   // COMANDO DELLE USCITE SUL SOLLEVAMENTO RIBALTATORE
   // 
   REGION COMANDO DELLE USCITE SOLLEVATORE RIBALTA P3
       // Sollevatore Ribalta Semi guscio prodotto Stazione P3 - RIPOSO
       "A0301_CinghiaTrasporto_1.1_V_Rest_1":= "A0301_Ribaltatore".Solleva_Rib[1].DataOut.RestSolenoid;
       "A0301_CinghiaTrasporto_2.1_V_Rest_1" := "A0301_Ribaltatore".Solleva_Rib[2].DataOut.RestSolenoid;
       "A0301_CinghiaTrasporto_3.1_V_Rest_1" := "A0301_Ribaltatore".Solleva_Rib[3].DataOut.RestSolenoid;
       "A0301_CinghiaTrasporto_4.1_V_Rest_1"  := "A0301_Ribaltatore".Solleva_Rib[4].DataOut.RestSolenoid;
       "A0301_CinghiaTrasporto_5.1_V_Rest_1" := "A0301_Ribaltatore".Solleva_Rib[5].DataOut.RestSolenoid;
       "A0301_CinghiaTrasporto_6.1_V_Rest_1" := "A0301_Ribaltatore".Solleva_Rib[6].DataOut.RestSolenoid;

       // Sollevatore Ribalta Semi guscio prodotto Stazione P3 - LAVORO
       "A0301_CinghiaTrasporto_1.1_V_Work_2":= "A0301_Ribaltatore".Solleva_Rib[1].DataOut.WorkSolenoid;
       "A0301_CinghiaTrasporto_2.1_V_Work_2" := "A0301_Ribaltatore".Solleva_Rib[2].DataOut.WorkSolenoid;
       "A0301_CinghiaTrasporto_3.1_V_Work_2" := "A0301_Ribaltatore".Solleva_Rib[3].DataOut.WorkSolenoid;
       "A0301_CinghiaTrasporto_4.1_V_Work_2" := "A0301_Ribaltatore".Solleva_Rib[4].DataOut.WorkSolenoid;
       "A0301_CinghiaTrasporto_5.1_V_Work_2" := "A0301_Ribaltatore".Solleva_Rib[5].DataOut.WorkSolenoid;
       "A0301_CinghiaTrasporto_6.1_V_Work_2":= "A0301_Ribaltatore".Solleva_Rib[6].DataOut.WorkSolenoid;

   END_REGION;
END_REGION
END_FUNCTION

FUNCTION_BLOCK "A0301_Ribaltatore_FB"   // FB60, LAD
TITLE = == GESTIONE DELLA STAZIONE RIBALTATORE ==
// stored: MemoryReserve 100, SetENOAutomatically false
   VAR_INPUT
      AreaInterface : "AreaInterface";
      ZSI : "udt_ZoneSafetyInterface";
      DSI_Feed : "udt_DeviceSafetyInterface";
      DSI_Valve : "udt_DeviceSafetyInterface";
      Drive : "TAx_DriveInterface";
      DataIn : Struct
         OP_MoveToPos_PB : Bool;
         OP_Rest_PB : Bool;
         OP_Work_PB : Bool;
      END_STRUCT;
      CIn { ExternalAccessible := 'False'; ExternalVisible := 'False'; ExternalWritable := 'False'} : Struct
         Manager : Struct
            Ax : "Positioning_EPOS_Machine_Manager";
            Solleva : "ValveMachine_Manager";
         END_STRUCT;
         SemiAut_PB : Bool;
         Ax_Req : Struct
            Pos0 : Bool;
            Pos1 : Bool;
            Pos2 : Bool;
            Pos3 : Bool;
         END_STRUCT;
         P2 : Struct
            Fermi : "ValveMachine_COut";
            Sollevatore : "ValveMachine_COut";
         END_STRUCT;
         P3 : Struct
            Fermi : "ValveMachine_COut";
         END_STRUCT;
         P4 : Struct
            Fermi : "ValveMachine_COut";
         END_STRUCT;
         Trasporto : "SpeedMachine_COut";
      END_STRUCT;
      Config : Struct
         Ax : "Positioning_EPOS_Machine_Config_NEW";
         Solleva_Rib : Array[1..6] of "ValveMachine_Config";
      END_STRUCT;
      HWID_Ax_TEL111 : HW_SUBMODULE;
   END_VAR
   VAR_OUTPUT
      MachineInterface { ExternalAccessible := 'False'; ExternalVisible := 'False'; ExternalWritable := 'False'} : "MachineInterface";
      DataOut : "Positioning_EPOS_Machine_DataOut";
      COut : Struct
         Solleva_Rib : "ValveMachine_COut";
         Ribaltatore : "Positioning_EPOS_Machine_COut";
         Ribaltatore_Sts : Struct
            Pos0_Reached : Bool;
            Pos1_Reached : Bool;
            Pos2_Reached : Bool;
            Pos3_Reached : Bool;
         END_STRUCT;
         Ribaltatore_AtRest : Bool;
      END_STRUCT;
   END_VAR
   VAR_IN_OUT
      Par_Manu : "Positioning_EPOS_Machine_Par";
      Par_Aut : "A0301_Mach_Ribaltatore_Par";
      Pers_Data : Struct
         EncoderAbsolute_Preset_OK : Bool;
         Persistent_ActualPosition : LReal;
      END_STRUCT;
   END_VAR
   VAR
      Alarm : Struct
         Solleva_Rib { S7_SetPoint := 'True'} : Array[1..6] of "ValveAlr";
         Ax { ExternalVisible := 'False'} : "Positioning_EPOS_Machine_Alr";
      END_STRUCT;
      Warning : Struct
         Ax { S7_SetPoint := 'True'} : "Positioning_EPOS_Machine_Wng";
         Solleva_Rib { S7_SetPoint := 'True'} : Array[1..6] of "ValveMachine_Wng";
         OP_REST_MissingCnd : Bool;   // Mancanza comando arresto
         OP_WORK_MissingCnd : Bool;   // Mancanza consenso lavoro
      END_STRUCT;
      ValueVelOvr { ExternalAccessible := 'False'; ExternalVisible := 'False'; ExternalWritable := 'False'} : Array[1..10] of Real;
      Ax : "Positioning_EPOS_Machine_FB_NEW";
      Solleva_Rib { S7_SetPoint := 'True'} : Array[1..6] of "ValveMachine_FB";
      TON : Struct
         DelayPos1_SG : IEC_TIMER;   // Tempo ritardo in Pos1 per appoggio semi-guscio
      END_STRUCT;
      Sts : Struct
         ReadyForMove : Bool;   // Pronto al movimento
         OP_CanMoveFreely : Bool;
         OP_MoveToPos_Cnd : Bool;
         OP_Rest_Cnd : Bool;
         OP_Work_Cnd : Bool;
         Solleva_Rib_AlarmPresence : Bool;
      END_STRUCT;
      Ctrl : Struct
         Ribaltatore : Struct
            OP_MoveToPos : Bool;
            Ax_MoveToPos : Bool;
         END_STRUCT;
         Solleva : Struct
            OP_Rest_Man : Bool;
            OP_Work_Man : Bool;
            OP_Rest_Aut : Bool;
            OP_Work_Aut : Bool;
            OP_Rest : Bool;
            OP_Work : Bool;
         END_STRUCT;
      END_STRUCT;
      HMI : Struct
         Ax : Struct
            B_Preset : Bool;
            PresetPosition : LReal;
            TargetPosition : LReal;
         END_STRUCT;
         SollevaRibSts { S7_SetPoint := 'True'} : "UDT_HMI-Sts_ValvePosA0301";
         OP_Sel_Pos0 : Bool;
         OP_Sel_Pos1 : Bool;
         OP_Sel_Pos2 : Bool;
         OP_Sel_Pos3 : Bool;
      END_STRUCT;
      AUX : Struct
         Solleva_Rib : Struct
            OP_Rest_PB : Bool;
            OP_Work_PB : Bool;
         END_STRUCT;
         Ribaltatore : Struct
            Ax_MoveToPos_PB : Bool;
         END_STRUCT;
      END_STRUCT;
      TON_Anticipi : Struct
         Rest : Struct
            SollevaRib { S7_SetPoint := 'True'} : IEC_TIMER;
         END_STRUCT;
         Work : Struct
            SollevaRib : IEC_TIMER;
         END_STRUCT;
      END_STRUCT;
   END_VAR
   VAR_TEMP
      PE : Struct
         Solleva : Struct
            OP_Rest_PB : Bool;
            OP_Work_PB : Bool;
         END_STRUCT;
         Ribaltatore : Struct
            Ax_MoveToPos_PB : Bool;
         END_STRUCT;
      END_STRUCT;
      VelOvr_Max : Real;   // Velocità max trovata
      i : Int;
      Anticipi : Struct
         SollevaRib : Struct
            COut_Work : Bool;
            COut_Rest : Bool;
            Not_Ls_Work : Bool;
            Not_Ls_Rest : Bool;
         END_STRUCT;
      END_STRUCT;
      CheckAnticipo : Bool;
   END_VAR
   VAR_TEMP   // added for the SCL form of the ladder/FBD networks
      _w1 : Bool;
      _w2 : Bool;
      _w3 : Bool;
      _w4 : Bool;
      _w5 : Bool;
      _w6 : Bool;
      _w7 : Bool;
      _w8 : Bool;
      _w9 : Bool;
   END_VAR
BEGIN

REGION Network 2: Anticipi Movimento LAVORO
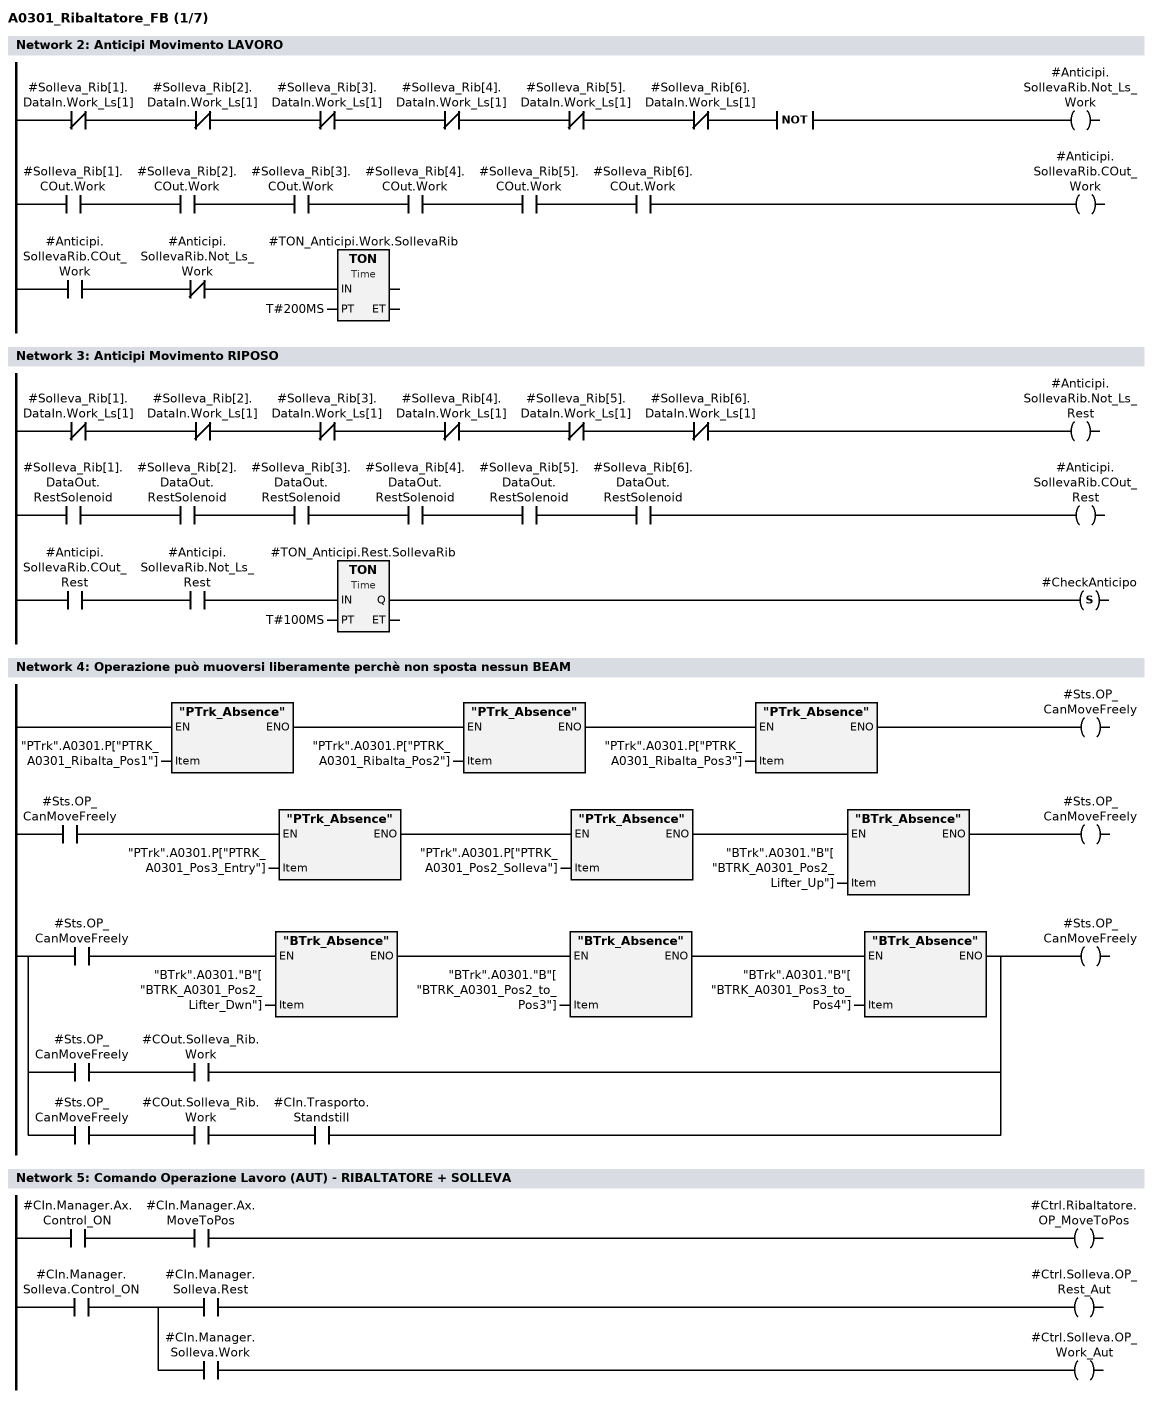
   RUNG wire#powerrail
      I_Contact( #Solleva_Rib[1].DataIn.Work_Ls[1] )
      I_Contact( #Solleva_Rib[2].DataIn.Work_Ls[1] )
      I_Contact( #Solleva_Rib[3].DataIn.Work_Ls[1] )
      I_Contact( #Solleva_Rib[4].DataIn.Work_Ls[1] )
      I_Contact( #Solleva_Rib[5].DataIn.Work_Ls[1] )
      I_Contact( #Solleva_Rib[6].DataIn.Work_Ls[1] )
      Not()
      Coil( #Anticipi.SollevaRib.Not_Ls_Work )
   END_RUNG
   RUNG wire#powerrail
      Contact( #Solleva_Rib[1].COut.Work )
      Contact( #Solleva_Rib[2].COut.Work )
      Contact( #Solleva_Rib[3].COut.Work )
      Contact( #Solleva_Rib[4].COut.Work )
      Contact( #Solleva_Rib[5].COut.Work )
      Contact( #Solleva_Rib[6].COut.Work )
      Coil( #Anticipi.SollevaRib.COut_Work )
   END_RUNG
   RUNG wire#powerrail
      Contact( #Anticipi.SollevaRib.COut_Work )
      I_Contact( #Anticipi.SollevaRib.Not_Ls_Work )
      { S7_Templates := "time_type := Time" } #TON_Anticipi.Work.SollevaRib.TON(pt := T#200MS, et =>)
   END_RUNG
   // the same network as SCL:
   #Anticipi.SollevaRib.Not_Ls_Work := NOT (NOT #Solleva_Rib[1].DataIn.Work_Ls[1] AND NOT #Solleva_Rib[2].DataIn.Work_Ls[1] AND NOT #Solleva_Rib[3].DataIn.Work_Ls[1] AND NOT #Solleva_Rib[4].DataIn.Work_Ls[1] AND NOT #Solleva_Rib[5].DataIn.Work_Ls[1] AND NOT #Solleva_Rib[6].DataIn.Work_Ls[1]);
   #Anticipi.SollevaRib.COut_Work := #Solleva_Rib[1].COut.Work AND #Solleva_Rib[2].COut.Work AND #Solleva_Rib[3].COut.Work AND #Solleva_Rib[4].COut.Work AND #Solleva_Rib[5].COut.Work AND #Solleva_Rib[6].COut.Work;
   #TON_Anticipi.Work.SollevaRib.TON(IN := #Anticipi.SollevaRib.COut_Work AND NOT #Anticipi.SollevaRib.Not_Ls_Work,
                           PT := T#200MS);
END_REGION

REGION Network 3: Anticipi Movimento RIPOSO
   RUNG wire#powerrail
      I_Contact( #Solleva_Rib[1].DataIn.Work_Ls[1] )
      I_Contact( #Solleva_Rib[2].DataIn.Work_Ls[1] )
      I_Contact( #Solleva_Rib[3].DataIn.Work_Ls[1] )
      I_Contact( #Solleva_Rib[4].DataIn.Work_Ls[1] )
      I_Contact( #Solleva_Rib[5].DataIn.Work_Ls[1] )
      I_Contact( #Solleva_Rib[6].DataIn.Work_Ls[1] )
      Coil( #Anticipi.SollevaRib.Not_Ls_Rest )
   END_RUNG
   RUNG wire#powerrail
      Contact( #Solleva_Rib[1].DataOut.RestSolenoid )
      Contact( #Solleva_Rib[2].DataOut.RestSolenoid )
      Contact( #Solleva_Rib[3].DataOut.RestSolenoid )
      Contact( #Solleva_Rib[4].DataOut.RestSolenoid )
      Contact( #Solleva_Rib[5].DataOut.RestSolenoid )
      Contact( #Solleva_Rib[6].DataOut.RestSolenoid )
      Coil( #Anticipi.SollevaRib.COut_Rest )
   END_RUNG
   RUNG wire#powerrail
      Contact( #Anticipi.SollevaRib.COut_Rest )
      Contact( #Anticipi.SollevaRib.Not_Ls_Rest )
      { S7_Templates := "time_type := Time" } #TON_Anticipi.Rest.SollevaRib.TON(pt := T#100MS, et =>)
      S_Coil( #CheckAnticipo )
   END_RUNG
   // the same network as SCL:
   #Anticipi.SollevaRib.Not_Ls_Rest := NOT #Solleva_Rib[1].DataIn.Work_Ls[1] AND NOT #Solleva_Rib[2].DataIn.Work_Ls[1] AND NOT #Solleva_Rib[3].DataIn.Work_Ls[1] AND NOT #Solleva_Rib[4].DataIn.Work_Ls[1] AND NOT #Solleva_Rib[5].DataIn.Work_Ls[1] AND NOT #Solleva_Rib[6].DataIn.Work_Ls[1];
   #Anticipi.SollevaRib.COut_Rest := #Solleva_Rib[1].DataOut.RestSolenoid AND #Solleva_Rib[2].DataOut.RestSolenoid AND #Solleva_Rib[3].DataOut.RestSolenoid AND #Solleva_Rib[4].DataOut.RestSolenoid AND #Solleva_Rib[5].DataOut.RestSolenoid AND #Solleva_Rib[6].DataOut.RestSolenoid;
   #TON_Anticipi.Rest.SollevaRib.TON(IN := #Anticipi.SollevaRib.COut_Rest AND #Anticipi.SollevaRib.Not_Ls_Rest,
                           PT := T#100MS);
   IF #TON_Anticipi.Rest.SollevaRib.Q THEN #CheckAnticipo := TRUE; END_IF;
END_REGION

REGION Network 4: Operazione può muoversi liberamente perchè non sposta nessun BEAM
   RUNG wire#powerrail
      "PTrk_Absence"(Item := "PTrk".A0301.P["PTRK_A0301_Ribalta_Pos1"])
      "PTrk_Absence"(Item := "PTrk".A0301.P["PTRK_A0301_Ribalta_Pos2"])
      "PTrk_Absence"(Item := "PTrk".A0301.P["PTRK_A0301_Ribalta_Pos3"])
      Coil( #Sts.OP_CanMoveFreely )
   END_RUNG
   RUNG wire#powerrail
      Contact( #Sts.OP_CanMoveFreely )
      "PTrk_Absence"(Item := "PTrk".A0301.P["PTRK_A0301_Pos3_Entry"])
      "PTrk_Absence"(Item := "PTrk".A0301.P["PTRK_A0301_Pos2_Solleva"])
      "BTrk_Absence"(Item := "BTrk".A0301."B"["BTRK_A0301_Pos2_Lifter_Up"])
      Coil( #Sts.OP_CanMoveFreely )
   END_RUNG
   RUNG wire#powerrail
      Contact( #Sts.OP_CanMoveFreely )
      "BTrk_Absence"(Item := "BTrk".A0301."B"["BTRK_A0301_Pos2_Lifter_Dwn"])
      "BTrk_Absence"(Item := "BTrk".A0301."B"["BTRK_A0301_Pos2_to_Pos3"])
      "BTrk_Absence"(Item := "BTrk".A0301."B"["BTRK_A0301_Pos3_to_Pos4"])
      wire#w1
      Coil( #Sts.OP_CanMoveFreely )
   END_RUNG
   RUNG wire#powerrail
      Contact( #Sts.OP_CanMoveFreely )
      Contact( #COut.Solleva_Rib.Work )
   END_RUNG wire#w1
   RUNG wire#powerrail
      Contact( #Sts.OP_CanMoveFreely )
      Contact( #COut.Solleva_Rib.Work )
      Contact( #CIn.Trasporto.Standstill )
   END_RUNG wire#w1
   // the same network as SCL:
   "PTrk_Absence"(Item := "PTrk".A0301.P["PTRK_A0301_Ribalta_Pos1"], ENO => #_w1);
   "PTrk_Absence"(EN := #_w1, Item := "PTrk".A0301.P["PTRK_A0301_Ribalta_Pos2"], ENO => #_w2);
   "PTrk_Absence"(EN := #_w2, Item := "PTrk".A0301.P["PTRK_A0301_Ribalta_Pos3"], ENO => #_w3);
   #Sts.OP_CanMoveFreely := #_w3;
   "PTrk_Absence"(EN := #Sts.OP_CanMoveFreely, Item := "PTrk".A0301.P["PTRK_A0301_Pos3_Entry"], ENO => #_w4);
   "PTrk_Absence"(EN := #_w4, Item := "PTrk".A0301.P["PTRK_A0301_Pos2_Solleva"], ENO => #_w5);
   "BTrk_Absence"(EN := #_w5, Item := "BTrk".A0301."B"["BTRK_A0301_Pos2_Lifter_Up"], ENO => #_w6);
   #Sts.OP_CanMoveFreely := #_w6;
   "BTrk_Absence"(EN := #Sts.OP_CanMoveFreely,
                  Item := "BTrk".A0301."B"["BTRK_A0301_Pos2_Lifter_Dwn"],
                  ENO => #_w7);
   "BTrk_Absence"(EN := #_w7, Item := "BTrk".A0301."B"["BTRK_A0301_Pos2_to_Pos3"], ENO => #_w8);
   "BTrk_Absence"(EN := #_w8, Item := "BTrk".A0301."B"["BTRK_A0301_Pos3_to_Pos4"], ENO => #_w9);
   #Sts.OP_CanMoveFreely := #_w9 OR (#Sts.OP_CanMoveFreely AND #COut.Solleva_Rib.Work) OR (#Sts.OP_CanMoveFreely AND #COut.Solleva_Rib.Work AND #CIn.Trasporto.Standstill);
END_REGION

REGION Network 5: Comando Operazione Lavoro (AUT) - RIBALTATORE + SOLLEVA
   RUNG wire#powerrail
      Contact( #CIn.Manager.Ax.Control_ON )
      Contact( #CIn.Manager.Ax.MoveToPos )
      Coil( #Ctrl.Ribaltatore.OP_MoveToPos )
   END_RUNG
   RUNG wire#powerrail
      Contact( #CIn.Manager.Solleva.Control_ON )
      wire#w1
      Contact( #CIn.Manager.Solleva.Rest )
      Coil( #Ctrl.Solleva.OP_Rest_Aut )
   END_RUNG
   RUNG wire#w1
      Contact( #CIn.Manager.Solleva.Work )
      Coil( #Ctrl.Solleva.OP_Work_Aut )
   END_RUNG
   // the same network as SCL:
   #Ctrl.Ribaltatore.OP_MoveToPos := #CIn.Manager.Ax.Control_ON AND #CIn.Manager.Ax.MoveToPos;
   #Ctrl.Solleva.OP_Rest_Aut := #CIn.Manager.Solleva.Control_ON AND #CIn.Manager.Solleva.Rest;
   #Ctrl.Solleva.OP_Work_Aut := #CIn.Manager.Solleva.Control_ON AND #CIn.Manager.Solleva.Work;
END_REGION

REGION Network 6: Comando Operazione Lavoro / Riposo (MAN) RIBALTATORE + SOLLEVA
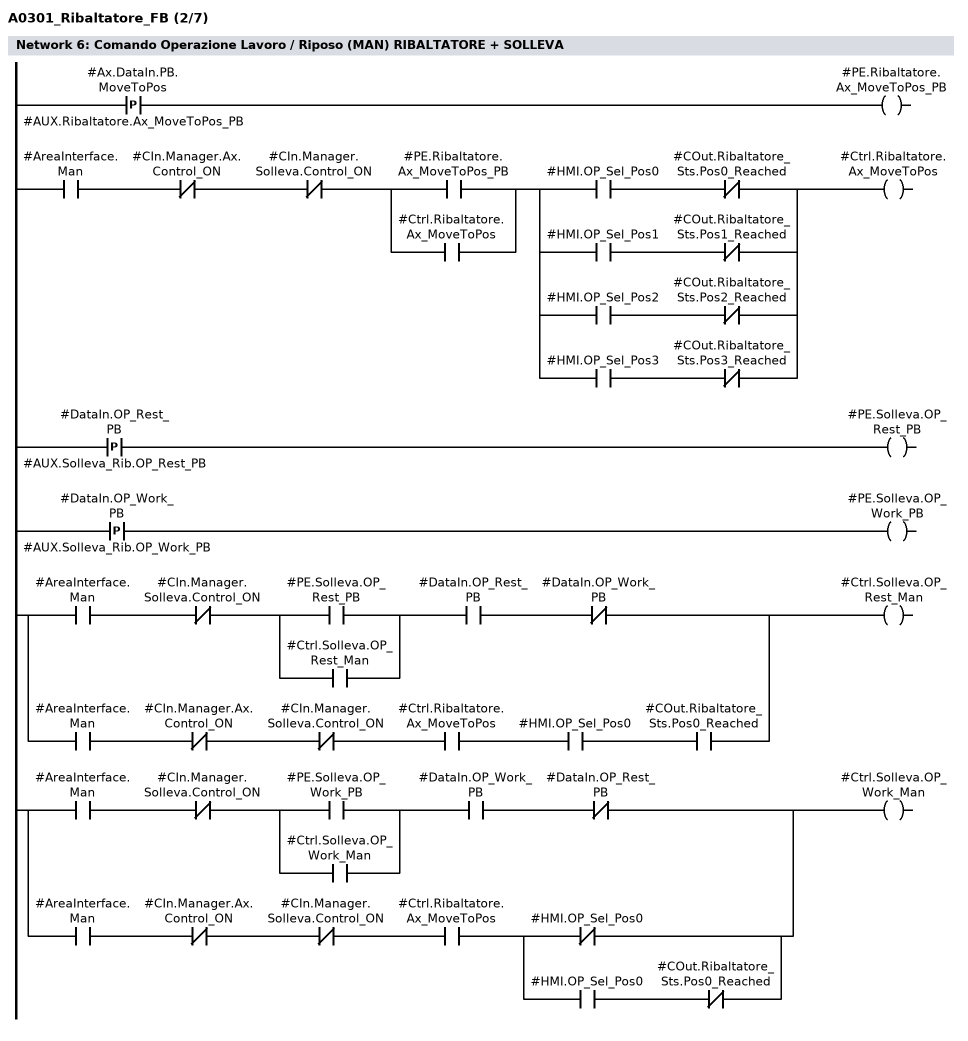
   RUNG wire#powerrail
      P_Contact(operand := #Ax.DataIn.PB.MoveToPos, bit := #AUX.Ribaltatore.Ax_MoveToPos_PB)
      Coil( #PE.Ribaltatore.Ax_MoveToPos_PB )
   END_RUNG
   RUNG wire#powerrail
      Contact( #AreaInterface.Man )
      I_Contact( #CIn.Manager.Ax.Control_ON )
      I_Contact( #CIn.Manager.Solleva.Control_ON )
      wire#w1
      Contact( #PE.Ribaltatore.Ax_MoveToPos_PB )
      wire#w2
      Contact( #HMI.OP_Sel_Pos0 )
      I_Contact( #COut.Ribaltatore_Sts.Pos0_Reached )
      wire#w3
      Coil( #Ctrl.Ribaltatore.Ax_MoveToPos )
   END_RUNG
   RUNG wire#w1
      Contact( #Ctrl.Ribaltatore.Ax_MoveToPos )
   END_RUNG wire#w2
   RUNG wire#w2
      Contact( #HMI.OP_Sel_Pos1 )
      I_Contact( #COut.Ribaltatore_Sts.Pos1_Reached )
   END_RUNG wire#w3
   RUNG wire#w2
      Contact( #HMI.OP_Sel_Pos2 )
      I_Contact( #COut.Ribaltatore_Sts.Pos2_Reached )
   END_RUNG wire#w3
   RUNG wire#w2
      Contact( #HMI.OP_Sel_Pos3 )
      I_Contact( #COut.Ribaltatore_Sts.Pos3_Reached )
   END_RUNG wire#w3
   RUNG wire#powerrail
      P_Contact(operand := #DataIn.OP_Rest_PB, bit := #AUX.Solleva_Rib.OP_Rest_PB)
      Coil( #PE.Solleva.OP_Rest_PB )
   END_RUNG
   RUNG wire#powerrail
      P_Contact(operand := #DataIn.OP_Work_PB, bit := #AUX.Solleva_Rib.OP_Work_PB)
      Coil( #PE.Solleva.OP_Work_PB )
   END_RUNG
   RUNG wire#powerrail
      Contact( #AreaInterface.Man )
      I_Contact( #CIn.Manager.Solleva.Control_ON )
      wire#w4
      Contact( #PE.Solleva.OP_Rest_PB )
      wire#w5
      Contact( #DataIn.OP_Rest_PB )
      I_Contact( #DataIn.OP_Work_PB )
      wire#w6
      Coil( #Ctrl.Solleva.OP_Rest_Man )
   END_RUNG
   RUNG wire#w4
      Contact( #Ctrl.Solleva.OP_Rest_Man )
   END_RUNG wire#w5
   RUNG wire#powerrail
      Contact( #AreaInterface.Man )
      I_Contact( #CIn.Manager.Ax.Control_ON )
      I_Contact( #CIn.Manager.Solleva.Control_ON )
      Contact( #Ctrl.Ribaltatore.Ax_MoveToPos )
      Contact( #HMI.OP_Sel_Pos0 )
      Contact( #COut.Ribaltatore_Sts.Pos0_Reached )
   END_RUNG wire#w6
   RUNG wire#powerrail
      Contact( #AreaInterface.Man )
      I_Contact( #CIn.Manager.Solleva.Control_ON )
      wire#w7
      Contact( #PE.Solleva.OP_Work_PB )
      wire#w8
      Contact( #DataIn.OP_Work_PB )
      I_Contact( #DataIn.OP_Rest_PB )
      wire#w9
      Coil( #Ctrl.Solleva.OP_Work_Man )
   END_RUNG
   RUNG wire#w7
      Contact( #Ctrl.Solleva.OP_Work_Man )
   END_RUNG wire#w8
   RUNG wire#powerrail
      Contact( #AreaInterface.Man )
      I_Contact( #CIn.Manager.Ax.Control_ON )
      I_Contact( #CIn.Manager.Solleva.Control_ON )
      Contact( #Ctrl.Ribaltatore.Ax_MoveToPos )
      wire#w10
      I_Contact( #HMI.OP_Sel_Pos0 )
   END_RUNG wire#w9
   RUNG wire#w10
      Contact( #HMI.OP_Sel_Pos0 )
      I_Contact( #COut.Ribaltatore_Sts.Pos0_Reached )
   END_RUNG wire#w9
   // the same network as SCL:
   #_w1 := #Ax.DataIn.PB.MoveToPos AND NOT #AUX.Ribaltatore.Ax_MoveToPos_PB;   // rising edge of #Ax.DataIn.PB.MoveToPos
   #AUX.Ribaltatore.Ax_MoveToPos_PB := #Ax.DataIn.PB.MoveToPos;
   #PE.Ribaltatore.Ax_MoveToPos_PB := #_w1;
   #Ctrl.Ribaltatore.Ax_MoveToPos := #AreaInterface.Man AND NOT #CIn.Manager.Ax.Control_ON AND NOT #CIn.Manager.Solleva.Control_ON AND (#PE.Ribaltatore.Ax_MoveToPos_PB OR #Ctrl.Ribaltatore.Ax_MoveToPos) AND ((#HMI.OP_Sel_Pos0 AND NOT #COut.Ribaltatore_Sts.Pos0_Reached) OR (#HMI.OP_Sel_Pos1 AND NOT #COut.Ribaltatore_Sts.Pos1_Reached) OR (#HMI.OP_Sel_Pos2 AND NOT #COut.Ribaltatore_Sts.Pos2_Reached) OR (#HMI.OP_Sel_Pos3 AND NOT #COut.Ribaltatore_Sts.Pos3_Reached));
   #_w2 := #DataIn.OP_Rest_PB AND NOT #AUX.Solleva_Rib.OP_Rest_PB;   // rising edge of #DataIn.OP_Rest_PB
   #AUX.Solleva_Rib.OP_Rest_PB := #DataIn.OP_Rest_PB;
   #PE.Solleva.OP_Rest_PB := #_w2;
   #_w3 := #DataIn.OP_Work_PB AND NOT #AUX.Solleva_Rib.OP_Work_PB;   // rising edge of #DataIn.OP_Work_PB
   #AUX.Solleva_Rib.OP_Work_PB := #DataIn.OP_Work_PB;
   #PE.Solleva.OP_Work_PB := #_w3;
   #Ctrl.Solleva.OP_Rest_Man := (#AreaInterface.Man AND NOT #CIn.Manager.Solleva.Control_ON AND (#PE.Solleva.OP_Rest_PB OR #Ctrl.Solleva.OP_Rest_Man) AND #DataIn.OP_Rest_PB AND NOT #DataIn.OP_Work_PB) OR (#AreaInterface.Man AND NOT #CIn.Manager.Ax.Control_ON AND NOT #CIn.Manager.Solleva.Control_ON AND #Ctrl.Ribaltatore.Ax_MoveToPos AND #HMI.OP_Sel_Pos0 AND #COut.Ribaltatore_Sts.Pos0_Reached);
   #Ctrl.Solleva.OP_Work_Man := (#AreaInterface.Man AND NOT #CIn.Manager.Solleva.Control_ON AND (#PE.Solleva.OP_Work_PB OR #Ctrl.Solleva.OP_Work_Man) AND #DataIn.OP_Work_PB AND NOT #DataIn.OP_Rest_PB) OR (#AreaInterface.Man AND NOT #CIn.Manager.Ax.Control_ON AND NOT #CIn.Manager.Solleva.Control_ON AND #Ctrl.Ribaltatore.Ax_MoveToPos AND (NOT #HMI.OP_Sel_Pos0 OR (#HMI.OP_Sel_Pos0 AND NOT #COut.Ribaltatore_Sts.Pos0_Reached)));
END_REGION

REGION Network 7: Condizioni movimento Operazione a Lavoro / Riposo
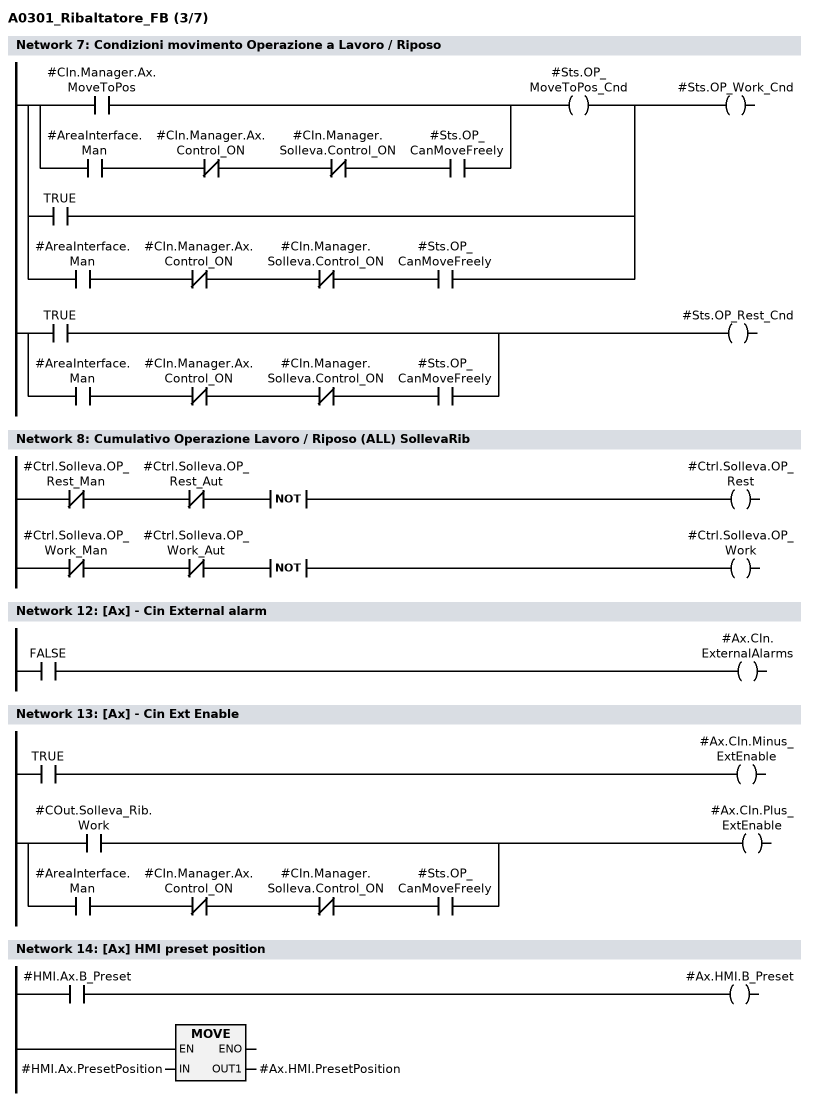
   RUNG wire#powerrail
      Contact( #CIn.Manager.Ax.MoveToPos )
      wire#w1
      Coil( #Sts.OP_MoveToPos_Cnd )
      wire#w2
      Coil( #Sts.OP_Work_Cnd )
   END_RUNG
   RUNG wire#powerrail
      Contact( #AreaInterface.Man )
      I_Contact( #CIn.Manager.Ax.Control_ON )
      I_Contact( #CIn.Manager.Solleva.Control_ON )
      Contact( #Sts.OP_CanMoveFreely )
   END_RUNG wire#w1
   RUNG wire#powerrail
      Contact( TRUE )
   END_RUNG wire#w2
   RUNG wire#powerrail
      Contact( #AreaInterface.Man )
      I_Contact( #CIn.Manager.Ax.Control_ON )
      I_Contact( #CIn.Manager.Solleva.Control_ON )
      Contact( #Sts.OP_CanMoveFreely )
   END_RUNG wire#w2
   RUNG wire#powerrail
      Contact( TRUE )
      wire#w3
      Coil( #Sts.OP_Rest_Cnd )
   END_RUNG
   RUNG wire#powerrail
      Contact( #AreaInterface.Man )
      I_Contact( #CIn.Manager.Ax.Control_ON )
      I_Contact( #CIn.Manager.Solleva.Control_ON )
      Contact( #Sts.OP_CanMoveFreely )
   END_RUNG wire#w3
   // the same network as SCL:
   #Sts.OP_MoveToPos_Cnd := #CIn.Manager.Ax.MoveToPos OR (#AreaInterface.Man AND NOT #CIn.Manager.Ax.Control_ON AND NOT #CIn.Manager.Solleva.Control_ON AND #Sts.OP_CanMoveFreely);
   #Sts.OP_Work_Cnd := #Sts.OP_MoveToPos_Cnd OR TRUE OR (#AreaInterface.Man AND NOT #CIn.Manager.Ax.Control_ON AND NOT #CIn.Manager.Solleva.Control_ON AND #Sts.OP_CanMoveFreely);
   #Sts.OP_Rest_Cnd := TRUE OR (#AreaInterface.Man AND NOT #CIn.Manager.Ax.Control_ON AND NOT #CIn.Manager.Solleva.Control_ON AND #Sts.OP_CanMoveFreely);
END_REGION

REGION Network 8: Cumulativo Operazione Lavoro / Riposo (ALL) SollevaRib
   RUNG wire#powerrail
      I_Contact( #Ctrl.Solleva.OP_Rest_Man )
      I_Contact( #Ctrl.Solleva.OP_Rest_Aut )
      Not()
      Coil( #Ctrl.Solleva.OP_Rest )
   END_RUNG
   RUNG wire#powerrail
      I_Contact( #Ctrl.Solleva.OP_Work_Man )
      I_Contact( #Ctrl.Solleva.OP_Work_Aut )
      Not()
      Coil( #Ctrl.Solleva.OP_Work )
   END_RUNG
   // the same network as SCL:
   #Ctrl.Solleva.OP_Rest := NOT (NOT #Ctrl.Solleva.OP_Rest_Man AND NOT #Ctrl.Solleva.OP_Rest_Aut);
   #Ctrl.Solleva.OP_Work := NOT (NOT #Ctrl.Solleva.OP_Work_Man AND NOT #Ctrl.Solleva.OP_Work_Aut);
END_REGION

REGION Network 9: <+>
END_REGION

REGION Network 10 (SCL): Solleva_Rib - Cin Manager (Esecuzione sequenza comandi)
   //
   #Solleva_Rib[1].Cin.Manager.Rest := FALSE;
   #Solleva_Rib[2].Cin.Manager.Rest := FALSE;
   #Solleva_Rib[3].Cin.Manager.Rest := FALSE;
   #Solleva_Rib[4].Cin.Manager.Rest := FALSE;
   #Solleva_Rib[5].Cin.Manager.Rest := FALSE;
   #Solleva_Rib[6].Cin.Manager.Rest := FALSE;

   //************************************
   #Solleva_Rib[1].Cin.Manager.Work := FALSE;
   #Solleva_Rib[2].Cin.Manager.Work := FALSE;
   #Solleva_Rib[3].Cin.Manager.Work := FALSE;
   #Solleva_Rib[4].Cin.Manager.Work := FALSE;
   #Solleva_Rib[5].Cin.Manager.Work := FALSE;
   #Solleva_Rib[6].Cin.Manager.Work := FALSE;

   //
   // CIn Manager  Control ON se ho un richiesta di comando attiva
   IF #AreaInterface.Aut OR #CIn.SemiAut_PB THEN
       #Solleva_Rib[1].Cin.Manager.Control_ON := TRUE;
       #Solleva_Rib[2].Cin.Manager.Control_ON := TRUE;
       #Solleva_Rib[3].Cin.Manager.Control_ON := TRUE;
       #Solleva_Rib[4].Cin.Manager.Control_ON := TRUE;
       #Solleva_Rib[5].Cin.Manager.Control_ON := TRUE;
       #Solleva_Rib[6].Cin.Manager.Control_ON := TRUE;
   ELSE
       #Solleva_Rib[1].Cin.Manager.Control_ON := FALSE;
       #Solleva_Rib[2].Cin.Manager.Control_ON := FALSE;
       #Solleva_Rib[3].Cin.Manager.Control_ON := FALSE;
       #Solleva_Rib[4].Cin.Manager.Control_ON := FALSE;
       #Solleva_Rib[5].Cin.Manager.Control_ON := FALSE;
       #Solleva_Rib[6].Cin.Manager.Control_ON := FALSE;
   END_IF;

   // Comando CIn Manager Work FERMI se Sfalsatore indietro
   IF #Ctrl.Solleva.OP_Work AND #Sts.OP_Work_Cnd THEN

       #Solleva_Rib[1].Cin.Manager.Work := TRUE;
       #Solleva_Rib[2].Cin.Manager.Work := TRUE;
       #Solleva_Rib[3].Cin.Manager.Work := TRUE;
       #Solleva_Rib[4].Cin.Manager.Work := TRUE;
       #Solleva_Rib[5].Cin.Manager.Work := TRUE;
       #Solleva_Rib[6].Cin.Manager.Work := TRUE;

   END_IF;

   // Comando CIn Manager Rest FERMI se Sfalsatore è basso
   IF #Ctrl.Solleva.OP_Rest AND #Sts.OP_Rest_Cnd THEN

       #Solleva_Rib[1].Cin.Manager.Rest := TRUE;
       #Solleva_Rib[2].Cin.Manager.Rest := TRUE;
       #Solleva_Rib[3].Cin.Manager.Rest := TRUE;
       #Solleva_Rib[4].Cin.Manager.Rest := TRUE;
       #Solleva_Rib[5].Cin.Manager.Rest := TRUE;
       #Solleva_Rib[6].Cin.Manager.Rest := TRUE;

   END_IF;
END_REGION

REGION Network 11 (SCL): RIFERIMENTI [AX] - Positioning Manager
   // ******************************************************************************************

       // Rampe in Manuale
       IF #AreaInterface.Man AND NOT #CIn.SemiAut_PB THEN
           #Ax.CIn.Manager.Acc := #Par_Manu.Man_Acc;
           #Ax.CIn.Manager.Dec := #Par_Manu.Man_Dec;
       END_IF;


   // ******************************************************************************************
   REGION // // CALCOLO DELLA VELOCITA' TRASFERITA DALL'IMPIANTO IN BASE ALLA LUNGHEZZA DEL PEZZO

       // Inizializzo variabile di appoggio controllo overide massimo a un valore basso rispetto setpoint
       IF "Sys".AuxFirstPLCCycle THEN
           #VelOvr_Max := 100.0;
       END_IF;

       // Trasferisco le varibili su un array
       #ValueVelOvr[1] := "PPrf_MAIN".ON_WORK.A0301_A0302.Ribaltatore.VelOvr_PLen_UpTo_1000;
       #ValueVelOvr[2] := "PPrf_MAIN".ON_WORK.A0301_A0302.Ribaltatore.VelOvr_PLen_UpTo_1500;
       #ValueVelOvr[3] := "PPrf_MAIN".ON_WORK.A0301_A0302.Ribaltatore.VelOvr_PLen_UpTo_2000;
       #ValueVelOvr[4] := "PPrf_MAIN".ON_WORK.A0301_A0302.Ribaltatore.VelOvr_PLen_UpTo_2500;
       #ValueVelOvr[5] := "PPrf_MAIN".ON_WORK.A0301_A0302.Ribaltatore.VelOvr_PLen_UpTo_3000;
       #ValueVelOvr[6] := "PPrf_MAIN".ON_WORK.A0301_A0302.Ribaltatore.VelOvr_PLen_UpTo_3500;
       #ValueVelOvr[7] := "PPrf_MAIN".ON_WORK.A0301_A0302.Ribaltatore.VelOvr_PLen_UpTo_4000;
       #ValueVelOvr[8] := "PPrf_MAIN".ON_WORK.A0301_A0302.Ribaltatore.VelOvr_PLen_UpTo_4500;
       #ValueVelOvr[9] := "PPrf_MAIN".ON_WORK.A0301_A0302.Ribaltatore.VelOvr_PLen_UpTo_5000;
       #ValueVelOvr[10] := "PPrf_MAIN".ON_WORK.A0301_A0302.Ribaltatore.VelOvr_PLen_UpTo_5500;

       // Ciclo per verificare la variabile maggiore per prenderla in lavoro
       FOR #i := 1 TO 10 DO
           IF #ValueVelOvr[#i] >= #VelOvr_Max THEN
               #VelOvr_Max := #ValueVelOvr[#i];
           END_IF;
       END_FOR;// 
   END_REGION ;

   IF #VelOvr_Max = 0.0 THEN
       #VelOvr_Max := 100.0;
   END_IF;

   // *****************************************************************************************
   REGION // CALCOLO DELLA VELOCITA' E TRASFERIMENTO IN BASE ALLO STATO IMPIANTO
       //
       #Ax.CIn.Manager := #CIn.Manager.Ax;
       //
       #Ax.CIn.VelocityOverride.Enable := TRUE;

       IF #Ax.CIn.Manager.Control_ON THEN
           // CALCOLO VELOCITA' IN BASE ALL'OVERIDE
           #Ax.CIn.VelocityOverride.Value := #VelOvr_Max;
       ELSE
           #Ax.CIn.VelocityOverride.Value := 100.0;
       END_IF;

   END_REGION ;
END_REGION

REGION Network 12: [Ax] - Cin External alarm
   RUNG wire#powerrail
      Contact( FALSE )
      Coil( #Ax.CIn.ExternalAlarms )
   END_RUNG
   // the same network as SCL:
   #Ax.CIn.ExternalAlarms := FALSE;
END_REGION

REGION Network 13: [Ax] - Cin Ext Enable
   RUNG wire#powerrail
      Contact( TRUE )
      Coil( #Ax.CIn.Minus_ExtEnable )
   END_RUNG
   RUNG wire#powerrail
      Contact( #COut.Solleva_Rib.Work )
      wire#w1
      Coil( #Ax.CIn.Plus_ExtEnable )
   END_RUNG
   RUNG wire#powerrail
      Contact( #AreaInterface.Man )
      I_Contact( #CIn.Manager.Ax.Control_ON )
      I_Contact( #CIn.Manager.Solleva.Control_ON )
      Contact( #Sts.OP_CanMoveFreely )
   END_RUNG wire#w1
   // the same network as SCL:
   #Ax.CIn.Minus_ExtEnable := TRUE;
   #Ax.CIn.Plus_ExtEnable := #COut.Solleva_Rib.Work OR (#AreaInterface.Man AND NOT #CIn.Manager.Ax.Control_ON AND NOT #CIn.Manager.Solleva.Control_ON AND #Sts.OP_CanMoveFreely);
END_REGION

REGION Network 14: [Ax] HMI preset position
   RUNG wire#powerrail
      Contact( #HMI.Ax.B_Preset )
      Coil( #Ax.HMI.B_Preset )
   END_RUNG
   RUNG wire#powerrail
      Move(in := #HMI.Ax.PresetPosition, out1 => #Ax.HMI.PresetPosition)
   END_RUNG
   // the same network as SCL:
   #Ax.HMI.B_Preset := #HMI.Ax.B_Preset;
   #Ax.HMI.PresetPosition := #HMI.Ax.PresetPosition;
END_REGION

REGION Network 15: [Ax] - Positioning Manager
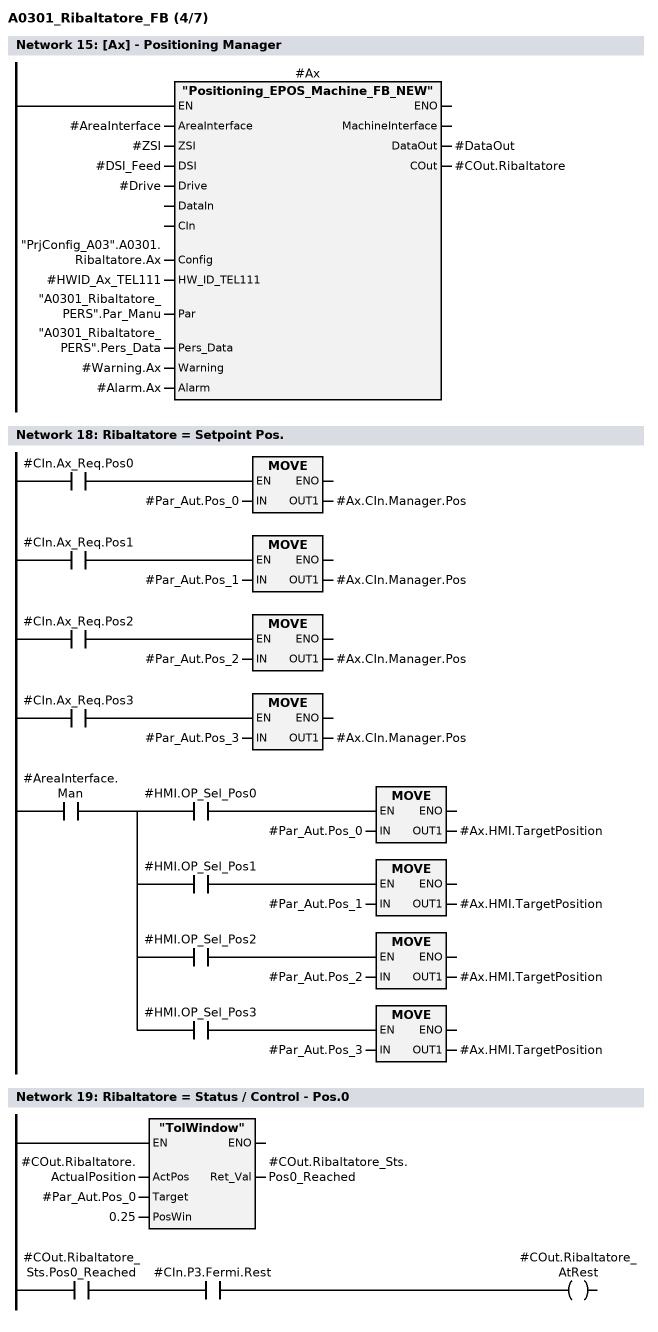
   RUNG wire#powerrail
      #Ax(AreaInterface := #AreaInterface, ZSI := #ZSI, DSI := #DSI_Feed, Drive := #Drive, DataIn :=, CIn :=, Config := "PrjConfig_A03".A0301.Ribaltatore.Ax, HW_ID_TEL111 := #HWID_Ax_TEL111, Par := "A0301_Ribaltatore_PERS".Par_Manu, Pers_Data := "A0301_Ribaltatore_PERS".Pers_Data, Warning := #Warning.Ax, Alarm := #Alarm.Ax, MachineInterface =>, DataOut => #DataOut, COut => #COut.Ribaltatore)
   END_RUNG
   // the same network as SCL:
   #Ax(AreaInterface := #AreaInterface,   // "Positioning_EPOS_Machine_FB_NEW"
       ZSI := #ZSI,
       DSI := #DSI_Feed,
       Drive := #Drive,
       Config := "PrjConfig_A03".A0301.Ribaltatore.Ax,
       HW_ID_TEL111 := #HWID_Ax_TEL111,
       Par := "A0301_Ribaltatore_PERS".Par_Manu,
       Pers_Data := "A0301_Ribaltatore_PERS".Pers_Data,
       Warning := #Warning.Ax,
       Alarm := #Alarm.Ax,
       DataOut => #DataOut,
       COut => #COut.Ribaltatore);
END_REGION

REGION Network 16: <+>
END_REGION

REGION Network 17: <<< CONTROLLO REQ da TRAKING E CAMBIO POS. >>>
END_REGION

REGION Network 18: Ribaltatore = Setpoint Pos.
   RUNG wire#powerrail
      Contact( #CIn.Ax_Req.Pos0 )
      Move(in := #Par_Aut.Pos_0, out1 => #Ax.CIn.Manager.Pos)
   END_RUNG
   RUNG wire#powerrail
      Contact( #CIn.Ax_Req.Pos1 )
      Move(in := #Par_Aut.Pos_1, out1 => #Ax.CIn.Manager.Pos)
   END_RUNG
   RUNG wire#powerrail
      Contact( #CIn.Ax_Req.Pos2 )
      Move(in := #Par_Aut.Pos_2, out1 => #Ax.CIn.Manager.Pos)
   END_RUNG
   RUNG wire#powerrail
      Contact( #CIn.Ax_Req.Pos3 )
      Move(in := #Par_Aut.Pos_3, out1 => #Ax.CIn.Manager.Pos)
   END_RUNG
   RUNG wire#powerrail
      Contact( #AreaInterface.Man )
      wire#w1
      Contact( #HMI.OP_Sel_Pos0 )
      Move(in := #Par_Aut.Pos_0, out1 => #Ax.HMI.TargetPosition)
   END_RUNG
   RUNG wire#w1
      Contact( #HMI.OP_Sel_Pos1 )
      Move(in := #Par_Aut.Pos_1, out1 => #Ax.HMI.TargetPosition)
   END_RUNG
   RUNG wire#w1
      Contact( #HMI.OP_Sel_Pos2 )
      Move(in := #Par_Aut.Pos_2, out1 => #Ax.HMI.TargetPosition)
   END_RUNG
   RUNG wire#w1
      Contact( #HMI.OP_Sel_Pos3 )
      Move(in := #Par_Aut.Pos_3, out1 => #Ax.HMI.TargetPosition)
   END_RUNG
   // the same network as SCL:
   IF #CIn.Ax_Req.Pos0 THEN #Ax.CIn.Manager.Pos := #Par_Aut.Pos_0; END_IF;
   IF #CIn.Ax_Req.Pos1 THEN #Ax.CIn.Manager.Pos := #Par_Aut.Pos_1; END_IF;
   IF #CIn.Ax_Req.Pos2 THEN #Ax.CIn.Manager.Pos := #Par_Aut.Pos_2; END_IF;
   IF #CIn.Ax_Req.Pos3 THEN #Ax.CIn.Manager.Pos := #Par_Aut.Pos_3; END_IF;
   IF #AreaInterface.Man AND #HMI.OP_Sel_Pos0 THEN #Ax.HMI.TargetPosition := #Par_Aut.Pos_0; END_IF;
   IF #AreaInterface.Man AND #HMI.OP_Sel_Pos1 THEN #Ax.HMI.TargetPosition := #Par_Aut.Pos_1; END_IF;
   IF #AreaInterface.Man AND #HMI.OP_Sel_Pos2 THEN #Ax.HMI.TargetPosition := #Par_Aut.Pos_2; END_IF;
   IF #AreaInterface.Man AND #HMI.OP_Sel_Pos3 THEN #Ax.HMI.TargetPosition := #Par_Aut.Pos_3; END_IF;
END_REGION

REGION Network 19: Ribaltatore = Status / Control - Pos.0
   RUNG wire#powerrail
      "TolWindow"(ActPos := #COut.Ribaltatore.ActualPosition, Target := #Par_Aut.Pos_0, PosWin := 0.25, Ret_Val => #COut.Ribaltatore_Sts.Pos0_Reached)
   END_RUNG
   RUNG wire#powerrail
      Contact( #COut.Ribaltatore_Sts.Pos0_Reached )
      Contact( #CIn.P3.Fermi.Rest )
      Coil( #COut.Ribaltatore_AtRest )
   END_RUNG
   // the same network as SCL:
   #COut.Ribaltatore_Sts.Pos0_Reached := "TolWindow"(ActPos := #COut.Ribaltatore.ActualPosition,
                           Target := #Par_Aut.Pos_0,
                           PosWin := 0.25);
   #COut.Ribaltatore_AtRest := #COut.Ribaltatore_Sts.Pos0_Reached AND #CIn.P3.Fermi.Rest;
END_REGION

REGION Network 20: Ribaltatore = Status / Control - Pos.1
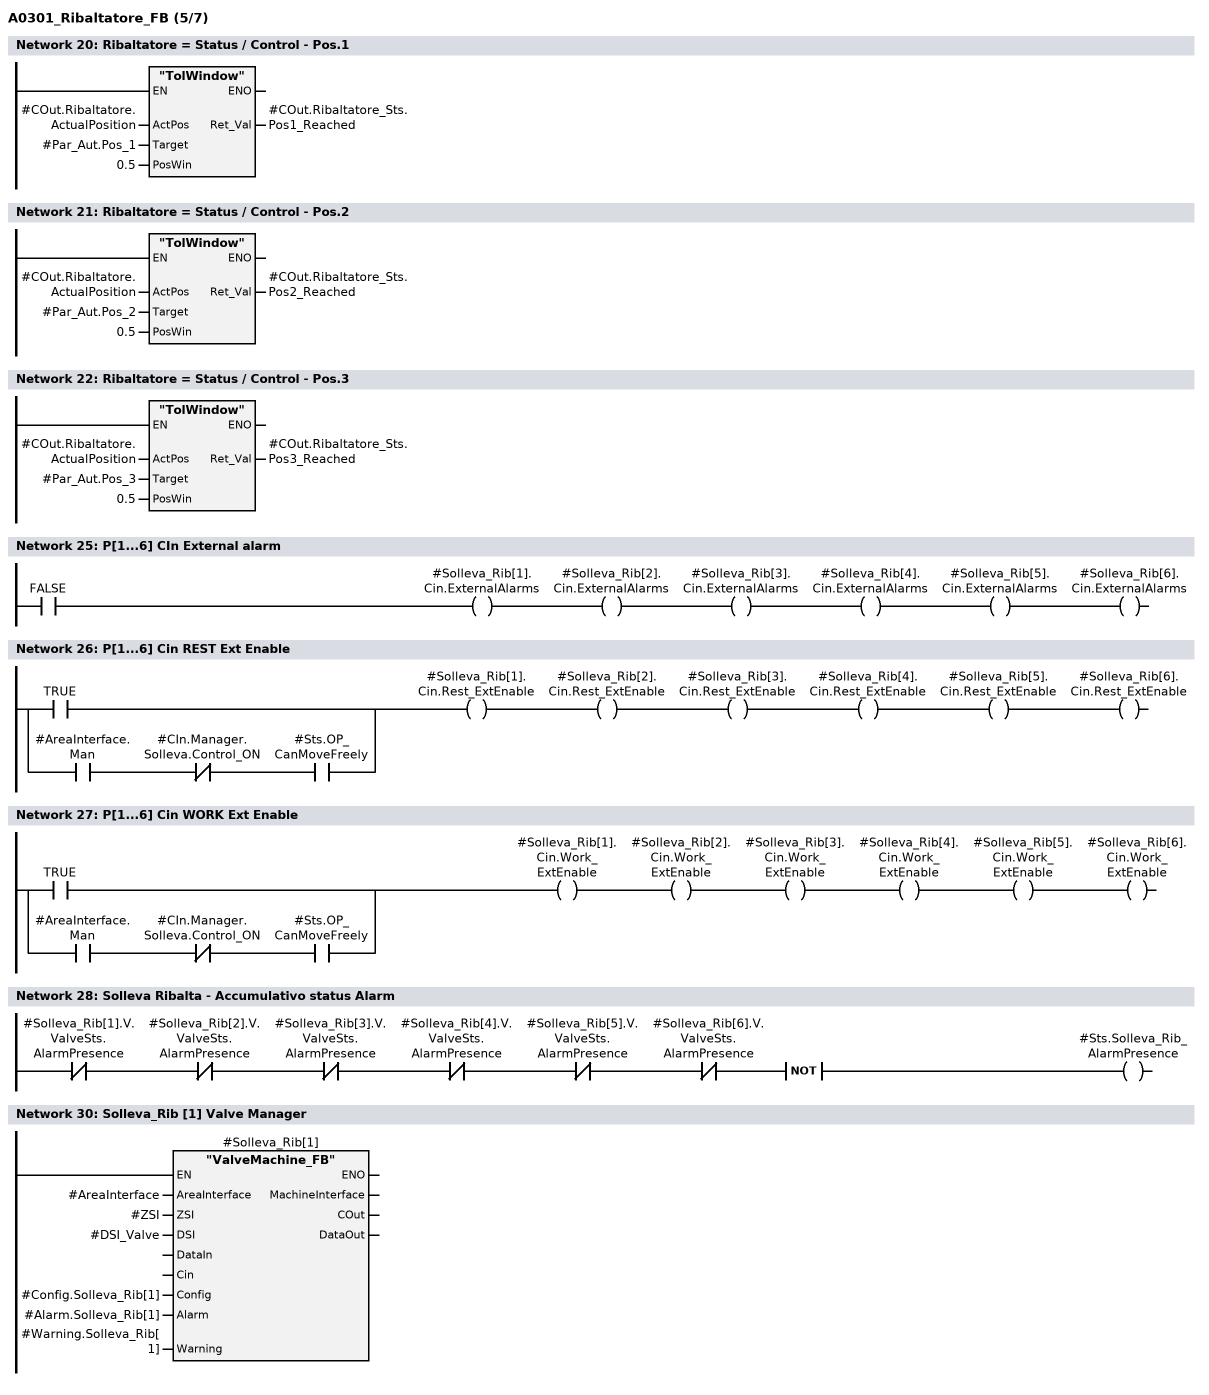
   RUNG wire#powerrail
      "TolWindow"(ActPos := #COut.Ribaltatore.ActualPosition, Target := #Par_Aut.Pos_1, PosWin := 0.5, Ret_Val => #COut.Ribaltatore_Sts.Pos1_Reached)
   END_RUNG
   // the same network as SCL:
   #COut.Ribaltatore_Sts.Pos1_Reached := "TolWindow"(ActPos := #COut.Ribaltatore.ActualPosition,
                           Target := #Par_Aut.Pos_1,
                           PosWin := 0.5);
END_REGION

REGION Network 21: Ribaltatore = Status / Control - Pos.2
   RUNG wire#powerrail
      "TolWindow"(ActPos := #COut.Ribaltatore.ActualPosition, Target := #Par_Aut.Pos_2, PosWin := 0.5, Ret_Val => #COut.Ribaltatore_Sts.Pos2_Reached)
   END_RUNG
   // the same network as SCL:
   #COut.Ribaltatore_Sts.Pos2_Reached := "TolWindow"(ActPos := #COut.Ribaltatore.ActualPosition,
                           Target := #Par_Aut.Pos_2,
                           PosWin := 0.5);
END_REGION

REGION Network 22: Ribaltatore = Status / Control - Pos.3
   RUNG wire#powerrail
      "TolWindow"(ActPos := #COut.Ribaltatore.ActualPosition, Target := #Par_Aut.Pos_3, PosWin := 0.5, Ret_Val => #COut.Ribaltatore_Sts.Pos3_Reached)
   END_RUNG
   // the same network as SCL:
   #COut.Ribaltatore_Sts.Pos3_Reached := "TolWindow"(ActPos := #COut.Ribaltatore.ActualPosition,
                           Target := #Par_Aut.Pos_3,
                           PosWin := 0.5);
END_REGION

REGION Network 23: <+>
END_REGION

REGION Network 24: << GESTIONE Solleva Ribalta >>
END_REGION

REGION Network 25: P[1...6] CIn External alarm
   RUNG wire#powerrail
      Contact( FALSE )
      Coil( #Solleva_Rib[1].Cin.ExternalAlarms )
      Coil( #Solleva_Rib[2].Cin.ExternalAlarms )
      Coil( #Solleva_Rib[3].Cin.ExternalAlarms )
      Coil( #Solleva_Rib[4].Cin.ExternalAlarms )
      Coil( #Solleva_Rib[5].Cin.ExternalAlarms )
      Coil( #Solleva_Rib[6].Cin.ExternalAlarms )
   END_RUNG
   // the same network as SCL:
   #Solleva_Rib[1].Cin.ExternalAlarms := FALSE;
   #Solleva_Rib[2].Cin.ExternalAlarms := FALSE;
   #Solleva_Rib[3].Cin.ExternalAlarms := FALSE;
   #Solleva_Rib[4].Cin.ExternalAlarms := FALSE;
   #Solleva_Rib[5].Cin.ExternalAlarms := FALSE;
   #Solleva_Rib[6].Cin.ExternalAlarms := FALSE;
END_REGION

REGION Network 26: P[1...6] Cin REST Ext Enable
   RUNG wire#powerrail
      Contact( TRUE )
      wire#w1
      Coil( #Solleva_Rib[1].Cin.Rest_ExtEnable )
      Coil( #Solleva_Rib[2].Cin.Rest_ExtEnable )
      Coil( #Solleva_Rib[3].Cin.Rest_ExtEnable )
      Coil( #Solleva_Rib[4].Cin.Rest_ExtEnable )
      Coil( #Solleva_Rib[5].Cin.Rest_ExtEnable )
      Coil( #Solleva_Rib[6].Cin.Rest_ExtEnable )
   END_RUNG
   RUNG wire#powerrail
      Contact( #AreaInterface.Man )
      I_Contact( #CIn.Manager.Solleva.Control_ON )
      Contact( #Sts.OP_CanMoveFreely )
   END_RUNG wire#w1
   // the same network as SCL:
   #Solleva_Rib[1].Cin.Rest_ExtEnable := TRUE OR (#AreaInterface.Man AND NOT #CIn.Manager.Solleva.Control_ON AND #Sts.OP_CanMoveFreely);
   #Solleva_Rib[2].Cin.Rest_ExtEnable := TRUE OR (#AreaInterface.Man AND NOT #CIn.Manager.Solleva.Control_ON AND #Sts.OP_CanMoveFreely);
   #Solleva_Rib[3].Cin.Rest_ExtEnable := TRUE OR (#AreaInterface.Man AND NOT #CIn.Manager.Solleva.Control_ON AND #Sts.OP_CanMoveFreely);
   #Solleva_Rib[4].Cin.Rest_ExtEnable := TRUE OR (#AreaInterface.Man AND NOT #CIn.Manager.Solleva.Control_ON AND #Sts.OP_CanMoveFreely);
   #Solleva_Rib[5].Cin.Rest_ExtEnable := TRUE OR (#AreaInterface.Man AND NOT #CIn.Manager.Solleva.Control_ON AND #Sts.OP_CanMoveFreely);
   #Solleva_Rib[6].Cin.Rest_ExtEnable := TRUE OR (#AreaInterface.Man AND NOT #CIn.Manager.Solleva.Control_ON AND #Sts.OP_CanMoveFreely);
END_REGION

REGION Network 27: P[1...6] Cin WORK Ext Enable
   RUNG wire#powerrail
      Contact( TRUE )
      wire#w1
      Coil( #Solleva_Rib[1].Cin.Work_ExtEnable )
      Coil( #Solleva_Rib[2].Cin.Work_ExtEnable )
      Coil( #Solleva_Rib[3].Cin.Work_ExtEnable )
      Coil( #Solleva_Rib[4].Cin.Work_ExtEnable )
      Coil( #Solleva_Rib[5].Cin.Work_ExtEnable )
      Coil( #Solleva_Rib[6].Cin.Work_ExtEnable )
   END_RUNG
   RUNG wire#powerrail
      Contact( #AreaInterface.Man )
      I_Contact( #CIn.Manager.Solleva.Control_ON )
      Contact( #Sts.OP_CanMoveFreely )
   END_RUNG wire#w1
   // the same network as SCL:
   #Solleva_Rib[1].Cin.Work_ExtEnable := TRUE OR (#AreaInterface.Man AND NOT #CIn.Manager.Solleva.Control_ON AND #Sts.OP_CanMoveFreely);
   #Solleva_Rib[2].Cin.Work_ExtEnable := TRUE OR (#AreaInterface.Man AND NOT #CIn.Manager.Solleva.Control_ON AND #Sts.OP_CanMoveFreely);
   #Solleva_Rib[3].Cin.Work_ExtEnable := TRUE OR (#AreaInterface.Man AND NOT #CIn.Manager.Solleva.Control_ON AND #Sts.OP_CanMoveFreely);
   #Solleva_Rib[4].Cin.Work_ExtEnable := TRUE OR (#AreaInterface.Man AND NOT #CIn.Manager.Solleva.Control_ON AND #Sts.OP_CanMoveFreely);
   #Solleva_Rib[5].Cin.Work_ExtEnable := TRUE OR (#AreaInterface.Man AND NOT #CIn.Manager.Solleva.Control_ON AND #Sts.OP_CanMoveFreely);
   #Solleva_Rib[6].Cin.Work_ExtEnable := TRUE OR (#AreaInterface.Man AND NOT #CIn.Manager.Solleva.Control_ON AND #Sts.OP_CanMoveFreely);
END_REGION

REGION Network 28: Solleva Ribalta - Accumulativo status Alarm
   RUNG wire#powerrail
      I_Contact( #Solleva_Rib[1].V.ValveSts.AlarmPresence )
      I_Contact( #Solleva_Rib[2].V.ValveSts.AlarmPresence )
      I_Contact( #Solleva_Rib[3].V.ValveSts.AlarmPresence )
      I_Contact( #Solleva_Rib[4].V.ValveSts.AlarmPresence )
      I_Contact( #Solleva_Rib[5].V.ValveSts.AlarmPresence )
      I_Contact( #Solleva_Rib[6].V.ValveSts.AlarmPresence )
      Not()
      Coil( #Sts.Solleva_Rib_AlarmPresence )
   END_RUNG
   // the same network as SCL:
   #Sts.Solleva_Rib_AlarmPresence := NOT (NOT #Solleva_Rib[1].V.ValveSts.AlarmPresence AND NOT #Solleva_Rib[2].V.ValveSts.AlarmPresence AND NOT #Solleva_Rib[3].V.ValveSts.AlarmPresence AND NOT #Solleva_Rib[4].V.ValveSts.AlarmPresence AND NOT #Solleva_Rib[5].V.ValveSts.AlarmPresence AND NOT #Solleva_Rib[6].V.ValveSts.AlarmPresence);
END_REGION

REGION Network 30: Solleva_Rib [1] Valve Manager
   RUNG wire#powerrail
      #Solleva_Rib[1](AreaInterface := #AreaInterface, ZSI := #ZSI, DSI := #DSI_Valve, DataIn :=, Cin :=, Config := #Config.Solleva_Rib[1], Alarm := #Alarm.Solleva_Rib[1], Warning := #Warning.Solleva_Rib[1], MachineInterface =>, COut =>, DataOut =>)
   END_RUNG
   // the same network as SCL:
   #Solleva_Rib[1](AreaInterface := #AreaInterface,   // "ValveMachine_FB"
                   ZSI := #ZSI,
                   DSI := #DSI_Valve,
                   Config := #Config.Solleva_Rib[1],
                   Alarm := #Alarm.Solleva_Rib[1],
                   Warning := #Warning.Solleva_Rib[1]);
END_REGION

REGION Network 31: Solleva_Rib [2] Valve Manager
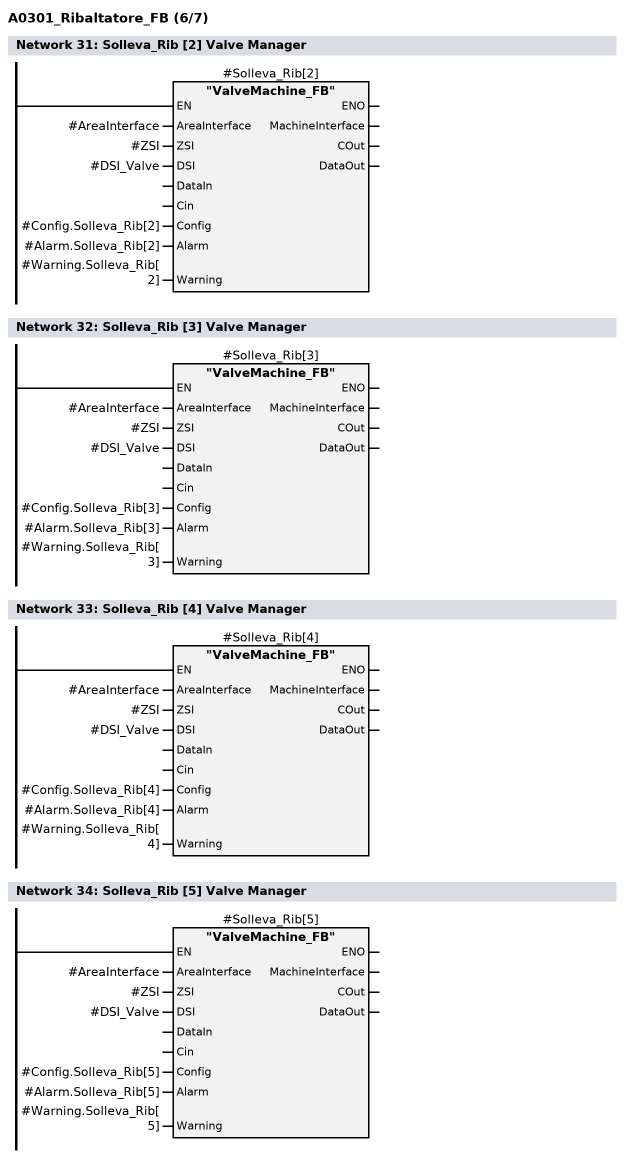
   RUNG wire#powerrail
      #Solleva_Rib[2](AreaInterface := #AreaInterface, ZSI := #ZSI, DSI := #DSI_Valve, DataIn :=, Cin :=, Config := #Config.Solleva_Rib[2], Alarm := #Alarm.Solleva_Rib[2], Warning := #Warning.Solleva_Rib[2], MachineInterface =>, COut =>, DataOut =>)
   END_RUNG
   // the same network as SCL:
   #Solleva_Rib[2](AreaInterface := #AreaInterface,   // "ValveMachine_FB"
                   ZSI := #ZSI,
                   DSI := #DSI_Valve,
                   Config := #Config.Solleva_Rib[2],
                   Alarm := #Alarm.Solleva_Rib[2],
                   Warning := #Warning.Solleva_Rib[2]);
END_REGION

REGION Network 32: Solleva_Rib [3] Valve Manager
   RUNG wire#powerrail
      #Solleva_Rib[3](AreaInterface := #AreaInterface, ZSI := #ZSI, DSI := #DSI_Valve, DataIn :=, Cin :=, Config := #Config.Solleva_Rib[3], Alarm := #Alarm.Solleva_Rib[3], Warning := #Warning.Solleva_Rib[3], MachineInterface =>, COut =>, DataOut =>)
   END_RUNG
   // the same network as SCL:
   #Solleva_Rib[3](AreaInterface := #AreaInterface,   // "ValveMachine_FB"
                   ZSI := #ZSI,
                   DSI := #DSI_Valve,
                   Config := #Config.Solleva_Rib[3],
                   Alarm := #Alarm.Solleva_Rib[3],
                   Warning := #Warning.Solleva_Rib[3]);
END_REGION

REGION Network 33: Solleva_Rib [4] Valve Manager
   RUNG wire#powerrail
      #Solleva_Rib[4](AreaInterface := #AreaInterface, ZSI := #ZSI, DSI := #DSI_Valve, DataIn :=, Cin :=, Config := #Config.Solleva_Rib[4], Alarm := #Alarm.Solleva_Rib[4], Warning := #Warning.Solleva_Rib[4], MachineInterface =>, COut =>, DataOut =>)
   END_RUNG
   // the same network as SCL:
   #Solleva_Rib[4](AreaInterface := #AreaInterface,   // "ValveMachine_FB"
                   ZSI := #ZSI,
                   DSI := #DSI_Valve,
                   Config := #Config.Solleva_Rib[4],
                   Alarm := #Alarm.Solleva_Rib[4],
                   Warning := #Warning.Solleva_Rib[4]);
END_REGION

REGION Network 34: Solleva_Rib [5] Valve Manager
   RUNG wire#powerrail
      #Solleva_Rib[5](AreaInterface := #AreaInterface, ZSI := #ZSI, DSI := #DSI_Valve, DataIn :=, Cin :=, Config := #Config.Solleva_Rib[5], Alarm := #Alarm.Solleva_Rib[5], Warning := #Warning.Solleva_Rib[5], MachineInterface =>, COut =>, DataOut =>)
   END_RUNG
   // the same network as SCL:
   #Solleva_Rib[5](AreaInterface := #AreaInterface,   // "ValveMachine_FB"
                   ZSI := #ZSI,
                   DSI := #DSI_Valve,
                   Config := #Config.Solleva_Rib[5],
                   Alarm := #Alarm.Solleva_Rib[5],
                   Warning := #Warning.Solleva_Rib[5]);
END_REGION

REGION Network 35: Solleva_Rib [6] Valve Manager
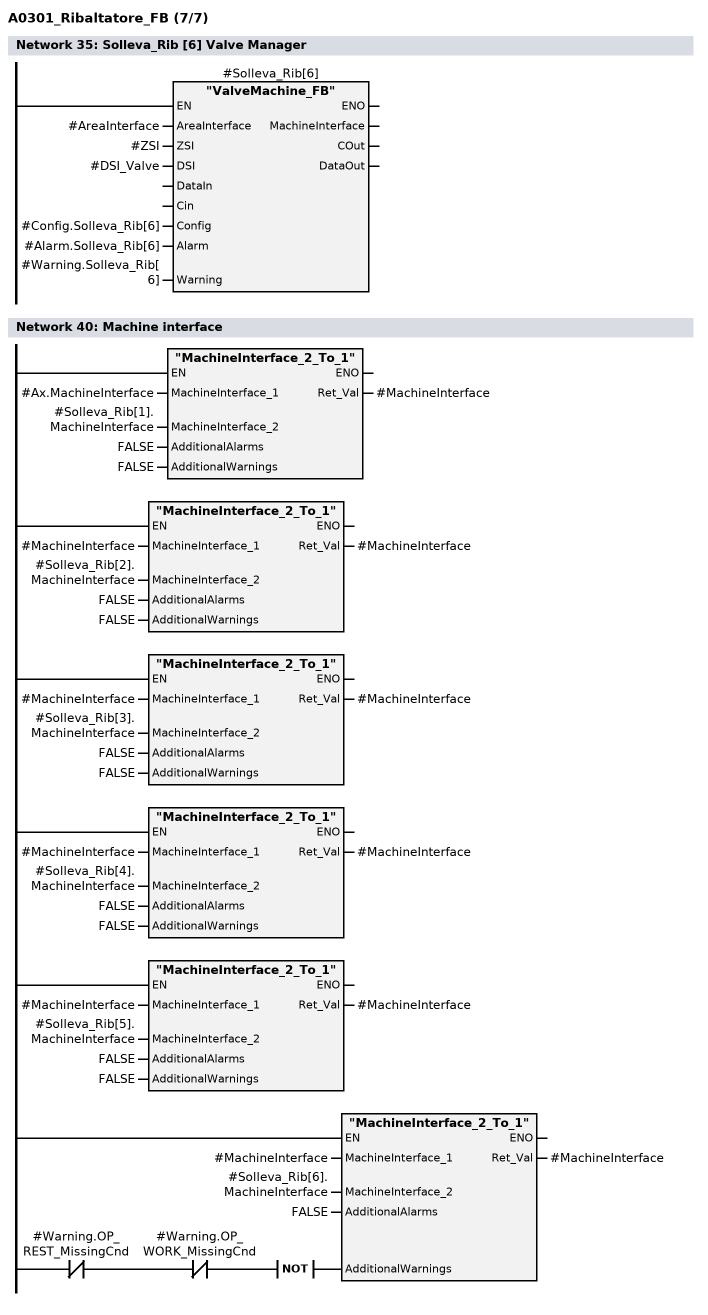
   RUNG wire#powerrail
      #Solleva_Rib[6](AreaInterface := #AreaInterface, ZSI := #ZSI, DSI := #DSI_Valve, DataIn :=, Cin :=, Config := #Config.Solleva_Rib[6], Alarm := #Alarm.Solleva_Rib[6], Warning := #Warning.Solleva_Rib[6], MachineInterface =>, COut =>, DataOut =>)
   END_RUNG
   // the same network as SCL:
   #Solleva_Rib[6](AreaInterface := #AreaInterface,   // "ValveMachine_FB"
                   ZSI := #ZSI,
                   DSI := #DSI_Valve,
                   Config := #Config.Solleva_Rib[6],
                   Alarm := #Alarm.Solleva_Rib[6],
                   Warning := #Warning.Solleva_Rib[6]);
END_REGION

REGION Network 36 (SCL): P[Solleva_Rib] COut
   #COut.Solleva_Rib.Standstill := FALSE;
   #COut.Solleva_Rib.Rest := FALSE;
   #COut.Solleva_Rib.Work := FALSE;

   REGION COut STANDSTILL Solleva_Rib
       // Controllo uscita COut STANDSTILL in base allo stato di tutti Solleva_Rib
       IF #Solleva_Rib[1].Sts.Standstill AND
           #Solleva_Rib[2].Sts.Standstill AND
           #Solleva_Rib[3].Sts.Standstill AND
           #Solleva_Rib[4].Sts.Standstill AND
           #Solleva_Rib[5].Sts.Standstill AND
           #Solleva_Rib[6].Sts.Standstill THEN
           #COut.Solleva_Rib.Standstill := TRUE;
       END_IF;
   END_REGION ;


   REGION COut AT REST Solleva_Rib

       // Controllo uscita COut AT_REST in base allo stato di tutti iSolleva_Rib
       IF  #Solleva_Rib[1].COut.Rest OR #TON_Anticipi.Rest.SollevaRib.Q AND
           #Solleva_Rib[2].COut.Rest OR #TON_Anticipi.Rest.SollevaRib.Q AND
           #Solleva_Rib[3].COut.Rest OR #TON_Anticipi.Rest.SollevaRib.Q AND
           #Solleva_Rib[4].COut.Rest OR #TON_Anticipi.Rest.SollevaRib.Q AND
           #Solleva_Rib[5].COut.Rest OR #TON_Anticipi.Rest.SollevaRib.Q AND
           #Solleva_Rib[6].COut.Rest OR #TON_Anticipi.Rest.SollevaRib.Q THEN
           #COut.Solleva_Rib.Rest := TRUE;
       END_IF;
   END_REGION ;

   REGION COut AT WORK Solleva_Rib
       // Controllo uscita COut AT_WORK in base allo stato di tutti i Solleva_Rib
       IF  #Solleva_Rib[1].COut.Work AND
           #Solleva_Rib[2].COut.Work AND
           #Solleva_Rib[3].COut.Work AND
           #Solleva_Rib[4].COut.Work AND
           #Solleva_Rib[5].COut.Work AND
           #Solleva_Rib[6].COut.Work THEN
           #COut.Solleva_Rib.Work := TRUE;
       END_IF;
   END_REGION ;
END_REGION

REGION Network 37: <+>
END_REGION

REGION Network 38 (SCL): HMI STATUS - Postazione
   // Area dati appoggio per HMI
   // SOLLEVA RIBALTA
   #HMI.SollevaRibSts.Standstill := #COut.Solleva_Rib.Standstill;
   #HMI.SollevaRibSts.Rest := #COut.Solleva_Rib.Rest;
   #HMI.SollevaRibSts.Work := #COut.Solleva_Rib.Work;
   #HMI.SollevaRibSts.AlarmPresence := #Sts.Solleva_Rib_AlarmPresence;
END_REGION

REGION Network 39: << MAIN MACHINE STATUS >>
END_REGION

REGION Network 40: Machine interface
   RUNG wire#powerrail
      "MachineInterface_2_To_1"(MachineInterface_1 := #Ax.MachineInterface, MachineInterface_2 := #Solleva_Rib[1].MachineInterface, AdditionalAlarms := FALSE, AdditionalWarnings := FALSE, Ret_Val => #MachineInterface)
   END_RUNG
   RUNG wire#powerrail
      "MachineInterface_2_To_1"(MachineInterface_1 := #MachineInterface, MachineInterface_2 := #Solleva_Rib[2].MachineInterface, AdditionalAlarms := FALSE, AdditionalWarnings := FALSE, Ret_Val => #MachineInterface)
   END_RUNG
   RUNG wire#powerrail
      "MachineInterface_2_To_1"(MachineInterface_1 := #MachineInterface, MachineInterface_2 := #Solleva_Rib[3].MachineInterface, AdditionalAlarms := FALSE, AdditionalWarnings := FALSE, Ret_Val => #MachineInterface)
   END_RUNG
   RUNG wire#powerrail
      "MachineInterface_2_To_1"(MachineInterface_1 := #MachineInterface, MachineInterface_2 := #Solleva_Rib[4].MachineInterface, AdditionalAlarms := FALSE, AdditionalWarnings := FALSE, Ret_Val => #MachineInterface)
   END_RUNG
   RUNG wire#powerrail
      "MachineInterface_2_To_1"(MachineInterface_1 := #MachineInterface, MachineInterface_2 := #Solleva_Rib[5].MachineInterface, AdditionalAlarms := FALSE, AdditionalWarnings := FALSE, Ret_Val => #MachineInterface)
   END_RUNG
   RUNG wire#powerrail
      "MachineInterface_2_To_1"(AdditionalWarnings := wire#w1, MachineInterface_1 := #MachineInterface, MachineInterface_2 := #Solleva_Rib[6].MachineInterface, AdditionalAlarms := FALSE, Ret_Val => #MachineInterface)
   END_RUNG
   RUNG wire#powerrail
      I_Contact( #Warning.OP_REST_MissingCnd )
      I_Contact( #Warning.OP_WORK_MissingCnd )
      Not()
   END_RUNG wire#w1
   // the same network as SCL:
   #MachineInterface := "MachineInterface_2_To_1"(MachineInterface_1 := #Ax.MachineInterface,
                           MachineInterface_2 := #Solleva_Rib[1].MachineInterface,
                           AdditionalAlarms := FALSE,
                           AdditionalWarnings := FALSE);
   #MachineInterface := "MachineInterface_2_To_1"(MachineInterface_1 := #MachineInterface,
                           MachineInterface_2 := #Solleva_Rib[2].MachineInterface,
                           AdditionalAlarms := FALSE,
                           AdditionalWarnings := FALSE);
   #MachineInterface := "MachineInterface_2_To_1"(MachineInterface_1 := #MachineInterface,
                           MachineInterface_2 := #Solleva_Rib[3].MachineInterface,
                           AdditionalAlarms := FALSE,
                           AdditionalWarnings := FALSE);
   #MachineInterface := "MachineInterface_2_To_1"(MachineInterface_1 := #MachineInterface,
                           MachineInterface_2 := #Solleva_Rib[4].MachineInterface,
                           AdditionalAlarms := FALSE,
                           AdditionalWarnings := FALSE);
   #MachineInterface := "MachineInterface_2_To_1"(MachineInterface_1 := #MachineInterface,
                           MachineInterface_2 := #Solleva_Rib[5].MachineInterface,
                           AdditionalAlarms := FALSE,
                           AdditionalWarnings := FALSE);
   #MachineInterface := "MachineInterface_2_To_1"(MachineInterface_1 := #MachineInterface,
                           MachineInterface_2 := #Solleva_Rib[6].MachineInterface,
                           AdditionalAlarms := FALSE,
                           AdditionalWarnings := NOT (NOT #Warning.OP_REST_MissingCnd AND NOT #Warning.OP_WORK_MissingCnd));
END_REGION
END_FUNCTION_BLOCK

FUNCTION "A0301_Fermi_P4_CALL" : Void   // FC121, LAD
// stored: SetENOAutomatically false
BEGIN

REGION Network 1 (SCL): << TRASFERIMENTO stati CIn del blocco >>
   // TRASFERIMENTO COMANDI #CIn MANAGER
   "A0301_Fermi_P4".CIn.Manager := "A0301_Manager".COut.P4.Fermi;
   //
   "A0301_Fermi_P4".CIn.SemiAut_Pb := "A0301_Manager".DataIn.SemiAut_Pb;

   // Trasferimento status alla Stazione P4 da COut a Cin delle stazioni successive
   "A0301_Fermi_P4".CIn.P3.Fermi := "A0301_Fermi_P3".COut.Fermi;

   // Trasferimenti status lettura posizioni Trasporto al Cin delle stazioni
   "A0301_Fermi_P3".CIn.Trasporto := "A0301_Trasporto".COut.Ax;
END_REGION

REGION Network 2 (SCL): << TRASFERIMENTO stati DataIn >>
   // "Sys".ByPass ===> SOSTITUIRE CON INGRESSI

   REGION TRASFERIMENTO DataIn DIGITAL INPUT dei LIMIT SWITCH
       // Trasferimento ingressi digitali Limit Switch Fermi P4
       // 
       "A0301_Fermi_P4".Fermi[1].DataIn.Rest_Ls[1] :="A0301_CinghiaTrasporto_1.2_Ls_Rest_3";
       "A0301_Fermi_P4".Fermi[2].DataIn.Rest_Ls[1] :="A0301_CinghiaTrasporto_2.2_Ls_Rest_3";
       "A0301_Fermi_P4".Fermi[3].DataIn.Rest_Ls[1] :="A0301_CinghiaTrasporto_3.2_Ls_Rest_3";
       "A0301_Fermi_P4".Fermi[4].DataIn.Rest_Ls[1] :="A0301_CinghiaTrasporto_4.2_Ls_Rest_3";
       "A0301_Fermi_P4".Fermi[5].DataIn.Rest_Ls[1] :="A0301_CinghiaTrasporto_5.2_Ls_Rest_3";
       "A0301_Fermi_P4".Fermi[6].DataIn.Rest_Ls[1] :="A0301_CinghiaTrasporto_6.2_Ls_Rest_3";

   END_REGION ;
END_REGION

REGION Network 3: DataIn - Fermi
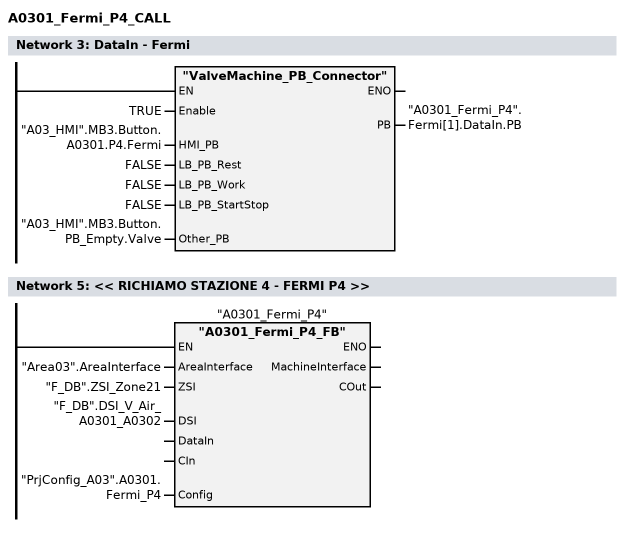
   RUNG wire#powerrail
      "ValveMachine_PB_Connector"(Enable := TRUE, HMI_PB := "A03_HMI".MB3.Button.A0301.P4.Fermi, LB_PB_Rest := FALSE, LB_PB_Work := FALSE, LB_PB_StartStop := FALSE, Other_PB := "A03_HMI".MB3.Button.PB_Empty.Valve, PB => "A0301_Fermi_P4".Fermi[1].DataIn.PB)
   END_RUNG
   // the same network as SCL:
   "ValveMachine_PB_Connector"(Enable := TRUE,
                           HMI_PB := "A03_HMI".MB3.Button.A0301.P4.Fermi,
                           LB_PB_Rest := FALSE,
                           LB_PB_Work := FALSE,
                           LB_PB_StartStop := FALSE,
                           Other_PB := "A03_HMI".MB3.Button.PB_Empty.Valve,
                           PB => "A0301_Fermi_P4".Fermi[1].DataIn.PB);
END_REGION

REGION Network 4 (SCL): DataIn - Fermi [1..6]
   // TRASFERIMENTO STATO PULSANTI - Comando manuale diretto 
   "A0301_Fermi_P4".Fermi[6].DataIn.PB.Rest := "A0301_Fermi_P4".Fermi[5].DataIn.PB.Rest := "A0301_Fermi_P4".Fermi[4].DataIn.PB.Rest :=
   "A0301_Fermi_P4".Fermi[3].DataIn.PB.Rest := "A0301_Fermi_P4".Fermi[2].DataIn.PB.Rest := "A0301_Fermi_P4".Fermi[1].DataIn.PB.Rest;

   "A0301_Fermi_P4".Fermi[6].DataIn.PB.Work := "A0301_Fermi_P4".Fermi[5].DataIn.PB.Work := "A0301_Fermi_P4".Fermi[4].DataIn.PB.Work :=
   "A0301_Fermi_P4".Fermi[3].DataIn.PB.Work := "A0301_Fermi_P4".Fermi[2].DataIn.PB.Work := "A0301_Fermi_P4".Fermi[1].DataIn.PB.Work;
END_REGION

REGION Network 5: << RICHIAMO STAZIONE 4 - FERMI P4 >>
   RUNG wire#powerrail
      "A0301_Fermi_P4"(AreaInterface := "Area03".AreaInterface, ZSI := "F_DB".ZSI_Zone21, DSI := "F_DB".DSI_V_Air_A0301_A0302, DataIn :=, CIn :=, Config := "PrjConfig_A03".A0301.Fermi_P4, MachineInterface =>, COut =>)
   END_RUNG
   // the same network as SCL:
   "A0301_Fermi_P4"(AreaInterface := "Area03".AreaInterface,   // "A0301_Fermi_P4_FB"
                    ZSI := "F_DB".ZSI_Zone21,
                    DSI := "F_DB".DSI_V_Air_A0301_A0302,
                    Config := "PrjConfig_A03".A0301.Fermi_P4);
END_REGION

REGION Network 6 (SCL): << TRASFERIMENTO stati DataOut >>
   // COLLEGARE LE USCITE DIGITALI
    REGION COMANDO DELLE USCITE FERMI P4

       // Fermi blocco prodotto Stazione P4 - RIPOSO

        "A0301_CinghiaTrasporto_1.2_V_Rest_3" := "A0301_Fermi_P4".Fermi[1].DataOut.RestSolenoid;
        "A0301_CinghiaTrasporto_2.2_V_Rest_3" := "A0301_Fermi_P4".Fermi[2].DataOut.RestSolenoid;
        "A0301_CinghiaTrasporto_3.2_V_Rest_3" := "A0301_Fermi_P4".Fermi[3].DataOut.RestSolenoid;
        "A0301_CinghiaTrasporto_4.2_V_Rest_3" := "A0301_Fermi_P4".Fermi[4].DataOut.RestSolenoid;
        "A0301_CinghiaTrasporto_5.2_V_Rest_3" := "A0301_Fermi_P4".Fermi[5].DataOut.RestSolenoid;
        "A0301_CinghiaTrasporto_6.2_V_Rest_3" := "A0301_Fermi_P4".Fermi[6].DataOut.RestSolenoid;

       // Fermi blocco prodotto Stazione P4 - LAVORO
       // 
        "A0301_CinghiaTrasporto_1.2_V_Work_4" := "A0301_Fermi_P4".Fermi[1].DataOut.WorkSolenoid;
        "A0301_CinghiaTrasporto_2.2_V_Work_4" := "A0301_Fermi_P4".Fermi[2].DataOut.WorkSolenoid;
        "A0301_CinghiaTrasporto_3.2_V_Work_4" := "A0301_Fermi_P4".Fermi[3].DataOut.WorkSolenoid;
        "A0301_CinghiaTrasporto_4.2_V_Work_4" := "A0301_Fermi_P4".Fermi[4].DataOut.WorkSolenoid;
        "A0301_CinghiaTrasporto_5.2_V_Work_4" := "A0301_Fermi_P4".Fermi[5].DataOut.WorkSolenoid;
        "A0301_CinghiaTrasporto_6.2_V_Work_4" := "A0301_Fermi_P4".Fermi[6].DataOut.WorkSolenoid;

   END_REGION ;
END_REGION
END_FUNCTION

FUNCTION_BLOCK "A0301_Fermi_P4_FB"   // FB67, LAD
TITLE = == GESTIONE DELLA STAZIONE P4 ==
// stored: MemoryReserve 100, SetENOAutomatically false
   VAR_INPUT
      AreaInterface : "AreaInterface";
      ZSI : "udt_ZoneSafetyInterface";
      DSI : "udt_DeviceSafetyInterface";
      DataIn : Struct
         OP_Rest_PB : Bool;
         OP_Work_PB : Bool;
      END_STRUCT;
      CIn : Struct
         Manager : "ValveMachine_Manager";
         SemiAut_Pb : Bool;
         P3 : Struct
            Fermi : "ValveMachine_COut";
         END_STRUCT;
         Trasporto : "SpeedMachine_COut";
      END_STRUCT;
      Config : Struct
         Fermi : Array[1..6] of "ValveMachine_Config";
         DelayMissingCondition : Time := T#3s;
      END_STRUCT;
   END_VAR
   VAR_OUTPUT
      MachineInterface : "MachineInterface";
      COut : Struct
         Fermi : "ValveMachine_COut";
      END_STRUCT;
   END_VAR
   VAR
      Alarm : Struct
         Fermi : Array[1..6] of "ValveAlr";
      END_STRUCT;
      Warning : Struct
         Fermi : Array[1..6] of "ValveMachine_Wng";
         OP_REST_MissingCnd : Bool;   // Mancanza comando arresto
         OP_WORK_MissingCnd : Bool;   // Mancanza consenso lavoro
      END_STRUCT;
      HMI : Struct
         Selection : Array[1..6] of Bool;   // 0=Disable / 1=Enable Pin
         FermiSts { S7_SetPoint := 'True'} : "UDT_HMI-Sts_ValvePosA0301";
      END_STRUCT;
      Sts : Struct
         Fermi_AlarmPresence : Bool;
         OP_CanMoveFreely : Bool;
         OP_Rest_Cnd : Bool;
         Op_Work_Cnd : Bool;
      END_STRUCT;
      Ctrl : Struct
         OP_Rest_Man : Bool;
         OP_Work_Man : Bool;
         OP_Rest_Aut : Bool;
         OP_Work_Aut : Bool;
         OP_Rest : Bool;
         OP_Work : Bool;
      END_STRUCT;
      Fermi { S7_SetPoint := 'True'} : Array[1..6] of "ValveMachine_FB";
      AUX : Struct
         OP_Rest_PB : Bool;
         OP_Work_PB : Bool;
      END_STRUCT;
      TON_OP_REST_MissingCnd { S7_SetPoint := 'True'} : TON_TIME;
      TON_OP_WORK_MissingCnd { S7_SetPoint := 'True'} : TON_TIME;
   END_VAR
   VAR_TEMP
      PE : Struct
         OP_Rest_PB : Bool;
         OP_Work_PB : Bool;
      END_STRUCT;
      Check : Struct
         Cndz1_P2_To_P4 : Bool;   // Check conditions to P4
         Cndz2_P2_To_P4 : Bool;
         Cndz1_Fermi_AtWork : Bool;
         Cndz2_Fermi_AtWork : Bool;
      END_STRUCT;
   END_VAR
   VAR_TEMP   // added for the SCL form of the ladder/FBD networks
      _w1 : Bool;
      _w2 : Bool;
      _w3 : Bool;
      _w4 : Bool;
   END_VAR
BEGIN

REGION Network 2: Operazione può muoversi liberamente perchè non sposta nessun BEAM
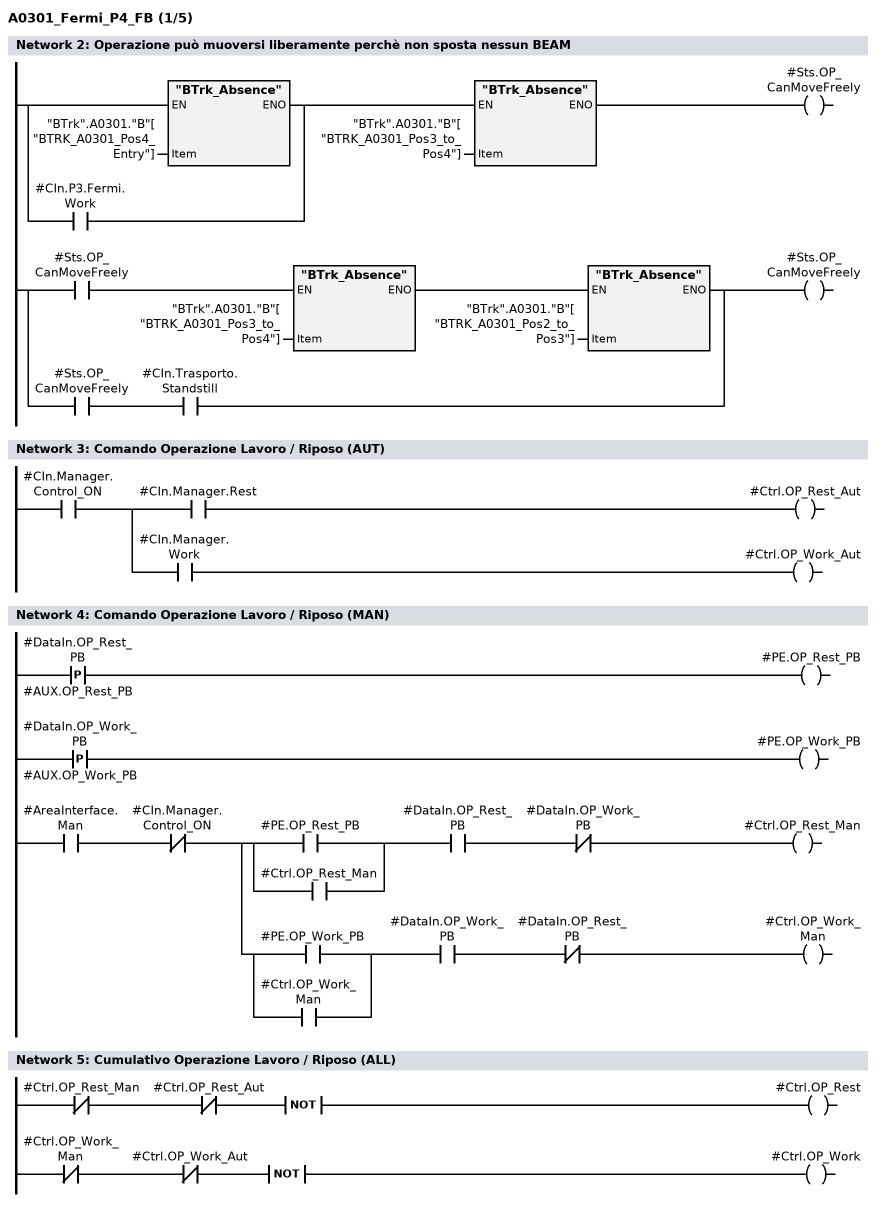
   RUNG wire#powerrail
      "BTrk_Absence"(Item := "BTrk".A0301."B"["BTRK_A0301_Pos4_Entry"])
      wire#w1
      "BTrk_Absence"(Item := "BTrk".A0301."B"["BTRK_A0301_Pos3_to_Pos4"])
      Coil( #Sts.OP_CanMoveFreely )
   END_RUNG
   RUNG wire#powerrail
      Contact( #CIn.P3.Fermi.Work )
   END_RUNG wire#w1
   RUNG wire#powerrail
      Contact( #Sts.OP_CanMoveFreely )
      "BTrk_Absence"(Item := "BTrk".A0301."B"["BTRK_A0301_Pos3_to_Pos4"])
      "BTrk_Absence"(Item := "BTrk".A0301."B"["BTRK_A0301_Pos2_to_Pos3"])
      wire#w2
      Coil( #Sts.OP_CanMoveFreely )
   END_RUNG
   RUNG wire#powerrail
      Contact( #Sts.OP_CanMoveFreely )
      Contact( #CIn.Trasporto.Standstill )
   END_RUNG wire#w2
   // the same network as SCL:
   "BTrk_Absence"(Item := "BTrk".A0301."B"["BTRK_A0301_Pos4_Entry"], ENO => #_w1);
   "BTrk_Absence"(EN := #_w1 OR #CIn.P3.Fermi.Work,
                  Item := "BTrk".A0301."B"["BTRK_A0301_Pos3_to_Pos4"],
                  ENO => #_w2);
   #Sts.OP_CanMoveFreely := #_w2;
   "BTrk_Absence"(EN := #Sts.OP_CanMoveFreely, Item := "BTrk".A0301."B"["BTRK_A0301_Pos3_to_Pos4"], ENO => #_w3);
   "BTrk_Absence"(EN := #_w3, Item := "BTrk".A0301."B"["BTRK_A0301_Pos2_to_Pos3"], ENO => #_w4);
   #Sts.OP_CanMoveFreely := #_w4 OR (#Sts.OP_CanMoveFreely AND #CIn.Trasporto.Standstill);
END_REGION

REGION Network 3: Comando Operazione Lavoro / Riposo (AUT)
   RUNG wire#powerrail
      Contact( #CIn.Manager.Control_ON )
      wire#w1
      Contact( #CIn.Manager.Rest )
      Coil( #Ctrl.OP_Rest_Aut )
   END_RUNG
   RUNG wire#w1
      Contact( #CIn.Manager.Work )
      Coil( #Ctrl.OP_Work_Aut )
   END_RUNG
   // the same network as SCL:
   #Ctrl.OP_Rest_Aut := #CIn.Manager.Control_ON AND #CIn.Manager.Rest;
   #Ctrl.OP_Work_Aut := #CIn.Manager.Control_ON AND #CIn.Manager.Work;
END_REGION

REGION Network 4: Comando Operazione Lavoro / Riposo (MAN)
   RUNG wire#powerrail
      P_Contact(operand := #DataIn.OP_Rest_PB, bit := #AUX.OP_Rest_PB)
      Coil( #PE.OP_Rest_PB )
   END_RUNG
   RUNG wire#powerrail
      P_Contact(operand := #DataIn.OP_Work_PB, bit := #AUX.OP_Work_PB)
      Coil( #PE.OP_Work_PB )
   END_RUNG
   RUNG wire#powerrail
      Contact( #AreaInterface.Man )
      I_Contact( #CIn.Manager.Control_ON )
      wire#w1
      Contact( #PE.OP_Rest_PB )
      wire#w2
      Contact( #DataIn.OP_Rest_PB )
      I_Contact( #DataIn.OP_Work_PB )
      Coil( #Ctrl.OP_Rest_Man )
   END_RUNG
   RUNG wire#w1
      Contact( #Ctrl.OP_Rest_Man )
   END_RUNG wire#w2
   RUNG wire#w1
      Contact( #PE.OP_Work_PB )
      wire#w3
      Contact( #DataIn.OP_Work_PB )
      I_Contact( #DataIn.OP_Rest_PB )
      Coil( #Ctrl.OP_Work_Man )
   END_RUNG
   RUNG wire#w1
      Contact( #Ctrl.OP_Work_Man )
   END_RUNG wire#w3
   // the same network as SCL:
   #_w1 := #DataIn.OP_Rest_PB AND NOT #AUX.OP_Rest_PB;   // rising edge of #DataIn.OP_Rest_PB
   #AUX.OP_Rest_PB := #DataIn.OP_Rest_PB;
   #PE.OP_Rest_PB := #_w1;
   #_w2 := #DataIn.OP_Work_PB AND NOT #AUX.OP_Work_PB;   // rising edge of #DataIn.OP_Work_PB
   #AUX.OP_Work_PB := #DataIn.OP_Work_PB;
   #PE.OP_Work_PB := #_w2;
   #_w3 := #AreaInterface.Man AND NOT #CIn.Manager.Control_ON;
   #Ctrl.OP_Rest_Man := #_w3 AND (#PE.OP_Rest_PB OR #Ctrl.OP_Rest_Man) AND #DataIn.OP_Rest_PB AND NOT #DataIn.OP_Work_PB;
   #Ctrl.OP_Work_Man := #_w3 AND (#PE.OP_Work_PB OR #Ctrl.OP_Work_Man) AND #DataIn.OP_Work_PB AND NOT #DataIn.OP_Rest_PB;
END_REGION

REGION Network 5: Cumulativo Operazione Lavoro / Riposo (ALL)
   RUNG wire#powerrail
      I_Contact( #Ctrl.OP_Rest_Man )
      I_Contact( #Ctrl.OP_Rest_Aut )
      Not()
      Coil( #Ctrl.OP_Rest )
   END_RUNG
   RUNG wire#powerrail
      I_Contact( #Ctrl.OP_Work_Man )
      I_Contact( #Ctrl.OP_Work_Aut )
      Not()
      Coil( #Ctrl.OP_Work )
   END_RUNG
   // the same network as SCL:
   #Ctrl.OP_Rest := NOT (NOT #Ctrl.OP_Rest_Man AND NOT #Ctrl.OP_Rest_Aut);
   #Ctrl.OP_Work := NOT (NOT #Ctrl.OP_Work_Man AND NOT #Ctrl.OP_Work_Aut);
END_REGION

REGION Network 6: Condizioni movimento Operazione a Lavoro / Riposo
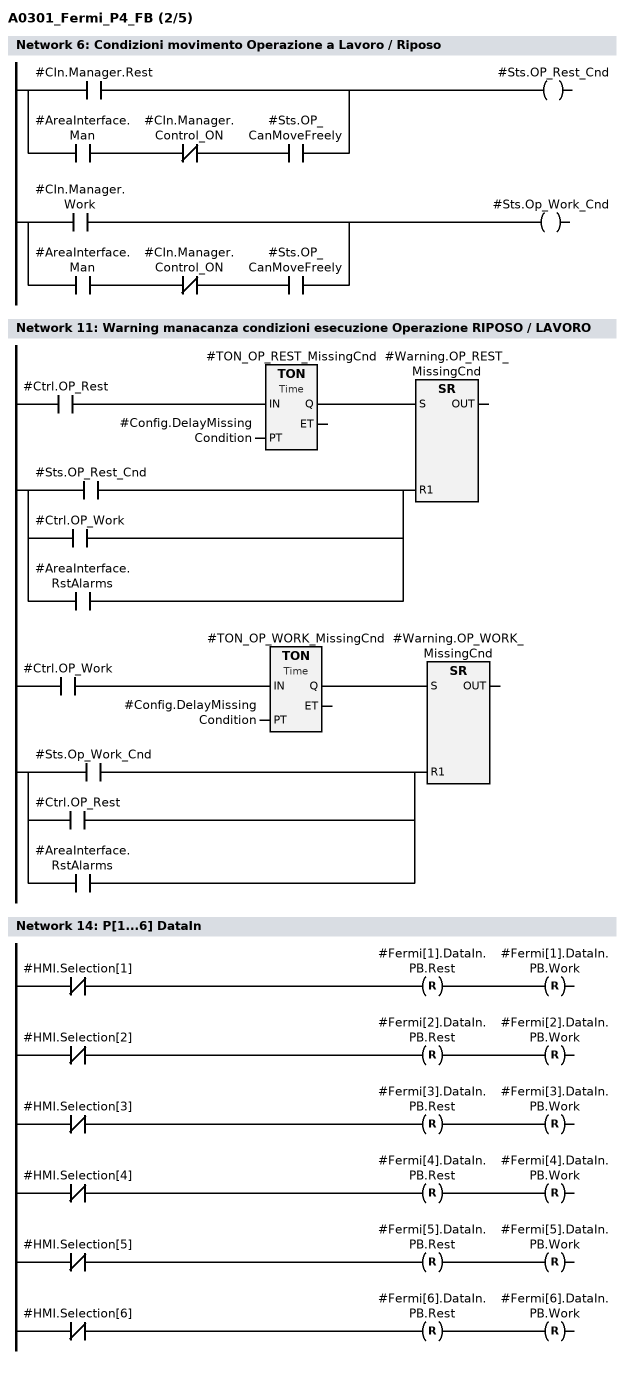
   RUNG wire#powerrail
      Contact( #CIn.Manager.Rest )
      wire#w1
      Coil( #Sts.OP_Rest_Cnd )
   END_RUNG
   RUNG wire#powerrail
      Contact( #AreaInterface.Man )
      I_Contact( #CIn.Manager.Control_ON )
      Contact( #Sts.OP_CanMoveFreely )
   END_RUNG wire#w1
   RUNG wire#powerrail
      Contact( #CIn.Manager.Work )
      wire#w2
      Coil( #Sts.Op_Work_Cnd )
   END_RUNG
   RUNG wire#powerrail
      Contact( #AreaInterface.Man )
      I_Contact( #CIn.Manager.Control_ON )
      Contact( #Sts.OP_CanMoveFreely )
   END_RUNG wire#w2
   // the same network as SCL:
   #Sts.OP_Rest_Cnd := #CIn.Manager.Rest OR (#AreaInterface.Man AND NOT #CIn.Manager.Control_ON AND #Sts.OP_CanMoveFreely);
   #Sts.Op_Work_Cnd := #CIn.Manager.Work OR (#AreaInterface.Man AND NOT #CIn.Manager.Control_ON AND #Sts.OP_CanMoveFreely);
END_REGION

REGION Network 7: <+>
END_REGION

REGION Network 8 (SCL): P[1...6] Cin Manager Comando arresto / lavoro
   //
   #Fermi[1].Cin.Manager.Rest := FALSE;
   #Fermi[2].Cin.Manager.Rest := FALSE;
   #Fermi[3].Cin.Manager.Rest := FALSE;
   #Fermi[4].Cin.Manager.Rest := FALSE;
   #Fermi[5].Cin.Manager.Rest := FALSE;
   #Fermi[6].Cin.Manager.Rest := FALSE;
   //************************************
   #Fermi[1].Cin.Manager.Work := FALSE;
   #Fermi[2].Cin.Manager.Work := FALSE;
   #Fermi[3].Cin.Manager.Work := FALSE;
   #Fermi[4].Cin.Manager.Work := FALSE;
   #Fermi[5].Cin.Manager.Work := FALSE;
   #Fermi[6].Cin.Manager.Work := FALSE;
   //
   // CIn Manager  Control ON se ho un richiesta di comando attiva
   IF #Ctrl.OP_Rest_Aut OR #Ctrl.OP_Work_Aut THEN
       #Fermi[1].Cin.Manager.Control_ON := TRUE;
       #Fermi[2].Cin.Manager.Control_ON := TRUE;
       #Fermi[3].Cin.Manager.Control_ON := TRUE;
       #Fermi[4].Cin.Manager.Control_ON := TRUE;
       #Fermi[5].Cin.Manager.Control_ON := TRUE;
       #Fermi[6].Cin.Manager.Control_ON := TRUE;
   ELSE
       #Fermi[1].Cin.Manager.Control_ON := FALSE;
       #Fermi[2].Cin.Manager.Control_ON := FALSE;
       #Fermi[3].Cin.Manager.Control_ON := FALSE;
       #Fermi[4].Cin.Manager.Control_ON := FALSE;
       #Fermi[5].Cin.Manager.Control_ON := FALSE;
       #Fermi[6].Cin.Manager.Control_ON := FALSE;
   END_IF;

   // CIn Manager Rest se ho un richiesta di comando arresto attiva
   IF #Ctrl.OP_Rest AND #Sts.OP_Rest_Cnd THEN

       #Fermi[1].Cin.Manager.Rest := TRUE;
       #Fermi[2].Cin.Manager.Rest := TRUE;
       #Fermi[3].Cin.Manager.Rest := TRUE;
       #Fermi[4].Cin.Manager.Rest := TRUE;
       #Fermi[5].Cin.Manager.Rest := TRUE;
       #Fermi[6].Cin.Manager.Rest := TRUE;

       // CIn Manager Work se ho un richiesta di comando lavoro attiva   
   ELSIF #Ctrl.OP_Work AND #Sts.Op_Work_Cnd THEN

       #Fermi[1].Cin.Manager.Work := TRUE;
       #Fermi[2].Cin.Manager.Work := TRUE;
       #Fermi[3].Cin.Manager.Work := TRUE;
       #Fermi[4].Cin.Manager.Work := TRUE;
       #Fermi[5].Cin.Manager.Work := TRUE;
       #Fermi[6].Cin.Manager.Work := TRUE;

   END_IF;
END_REGION

REGION Network 9 (SCL): P[1...6] CIn Abilitazioni Stop Manager
   //
   // CIn Manager Stop per richiesta apertura safety
   IF #CIn.Manager.EnableStopDoorOpeningReq THEN
       #Fermi[1].Cin.Manager.EnableStopDoorOpeningReq := TRUE;
       #Fermi[2].Cin.Manager.EnableStopDoorOpeningReq := TRUE;
       #Fermi[3].Cin.Manager.EnableStopDoorOpeningReq := TRUE;
       #Fermi[4].Cin.Manager.EnableStopDoorOpeningReq := TRUE;
       #Fermi[5].Cin.Manager.EnableStopDoorOpeningReq := TRUE;
       #Fermi[6].Cin.Manager.EnableStopDoorOpeningReq := TRUE;
   ELSE
       #Fermi[1].Cin.Manager.EnableStopDoorOpeningReq := FALSE;
       #Fermi[2].Cin.Manager.EnableStopDoorOpeningReq := FALSE;
       #Fermi[3].Cin.Manager.EnableStopDoorOpeningReq := FALSE;
       #Fermi[4].Cin.Manager.EnableStopDoorOpeningReq := FALSE;
       #Fermi[5].Cin.Manager.EnableStopDoorOpeningReq := FALSE;
       #Fermi[6].Cin.Manager.EnableStopDoorOpeningReq := FALSE;
   END_IF;
   // CIn Manager Stop in fase delle macchine precedenti
   IF #CIn.Manager.EnableStopInPhase THEN
       #Fermi[1].Cin.Manager.EnableStopInPhase := TRUE;
       #Fermi[2].Cin.Manager.EnableStopInPhase := TRUE;
       #Fermi[3].Cin.Manager.EnableStopInPhase := TRUE;
       #Fermi[4].Cin.Manager.EnableStopInPhase := TRUE;
       #Fermi[5].Cin.Manager.EnableStopInPhase := TRUE;
       #Fermi[6].Cin.Manager.EnableStopInPhase := TRUE;
   ELSE
       #Fermi[1].Cin.Manager.EnableStopInPhase := FALSE;
       #Fermi[2].Cin.Manager.EnableStopInPhase := FALSE;
       #Fermi[3].Cin.Manager.EnableStopInPhase := FALSE;
       #Fermi[4].Cin.Manager.EnableStopInPhase := FALSE;
       #Fermi[5].Cin.Manager.EnableStopInPhase := FALSE;
       #Fermi[6].Cin.Manager.EnableStopInPhase := FALSE;
   END_IF;

   // CIn Manager Stop programmato configurabile a piacere
   IF #CIn.Manager.EnableStopProgrammed THEN
       #Fermi[1].Cin.Manager.EnableStopProgrammed := TRUE;
       #Fermi[2].Cin.Manager.EnableStopProgrammed := TRUE;
       #Fermi[3].Cin.Manager.EnableStopProgrammed := TRUE;
       #Fermi[4].Cin.Manager.EnableStopProgrammed := TRUE;
       #Fermi[5].Cin.Manager.EnableStopProgrammed := TRUE;
       #Fermi[6].Cin.Manager.EnableStopProgrammed := TRUE;
   ELSE
       #Fermi[1].Cin.Manager.EnableStopProgrammed := FALSE;
       #Fermi[2].Cin.Manager.EnableStopProgrammed := FALSE;
       #Fermi[3].Cin.Manager.EnableStopProgrammed := FALSE;
       #Fermi[4].Cin.Manager.EnableStopProgrammed := FALSE;
       #Fermi[5].Cin.Manager.EnableStopProgrammed := FALSE;
       #Fermi[6].Cin.Manager.EnableStopProgrammed := FALSE;
   END_IF;
END_REGION

REGION Network 10: <+>
END_REGION

REGION Network 11: Warning manacanza condizioni esecuzione Operazione RIPOSO / LAVORO
   RUNG wire#powerrail
      Contact( #Ctrl.OP_Rest )
      { S7_Templates := "time_type := Time" } #TON_OP_REST_MissingCnd.TON(pt := #Config.DelayMissingCondition, et =>)
      S_SR(operand := #Warning.OP_REST_MissingCnd, r1 := wire#w1)
   END_RUNG
   RUNG wire#powerrail
      Contact( #Sts.OP_Rest_Cnd )
   END_RUNG wire#w1
   RUNG wire#powerrail
      Contact( #Ctrl.OP_Work )
   END_RUNG wire#w1
   RUNG wire#powerrail
      Contact( #AreaInterface.RstAlarms )
   END_RUNG wire#w1
   RUNG wire#powerrail
      Contact( #Ctrl.OP_Work )
      { S7_Templates := "time_type := Time" } #TON_OP_WORK_MissingCnd.TON(pt := #Config.DelayMissingCondition, et =>)
      S_SR(operand := #Warning.OP_WORK_MissingCnd, r1 := wire#w2)
   END_RUNG
   RUNG wire#powerrail
      Contact( #Sts.Op_Work_Cnd )
   END_RUNG wire#w2
   RUNG wire#powerrail
      Contact( #Ctrl.OP_Rest )
   END_RUNG wire#w2
   RUNG wire#powerrail
      Contact( #AreaInterface.RstAlarms )
   END_RUNG wire#w2
   // the same network as SCL:
   #TON_OP_REST_MissingCnd(IN := #Ctrl.OP_Rest, PT := #Config.DelayMissingCondition);   // TON
   IF #TON_OP_REST_MissingCnd.Q THEN
       #Warning.OP_REST_MissingCnd := TRUE;   // SR flip-flop
   END_IF;
   IF #Sts.OP_Rest_Cnd OR #Ctrl.OP_Work OR #AreaInterface.RstAlarms THEN
       #Warning.OP_REST_MissingCnd := FALSE;
   END_IF;
   #TON_OP_WORK_MissingCnd(IN := #Ctrl.OP_Work, PT := #Config.DelayMissingCondition);   // TON
   IF #TON_OP_WORK_MissingCnd.Q THEN
       #Warning.OP_WORK_MissingCnd := TRUE;   // SR flip-flop
   END_IF;
   IF #Sts.Op_Work_Cnd OR #Ctrl.OP_Rest OR #AreaInterface.RstAlarms THEN
       #Warning.OP_WORK_MissingCnd := FALSE;
   END_IF;
END_REGION

REGION Network 12: <+>
END_REGION

REGION Network 13: << GESTIONE FERMI >>
END_REGION

REGION Network 14: P[1...6] DataIn
   RUNG wire#powerrail
      I_Contact( #HMI.Selection[1] )
      R_Coil( #Fermi[1].DataIn.PB.Rest )
      R_Coil( #Fermi[1].DataIn.PB.Work )
   END_RUNG
   RUNG wire#powerrail
      I_Contact( #HMI.Selection[2] )
      R_Coil( #Fermi[2].DataIn.PB.Rest )
      R_Coil( #Fermi[2].DataIn.PB.Work )
   END_RUNG
   RUNG wire#powerrail
      I_Contact( #HMI.Selection[3] )
      R_Coil( #Fermi[3].DataIn.PB.Rest )
      R_Coil( #Fermi[3].DataIn.PB.Work )
   END_RUNG
   RUNG wire#powerrail
      I_Contact( #HMI.Selection[4] )
      R_Coil( #Fermi[4].DataIn.PB.Rest )
      R_Coil( #Fermi[4].DataIn.PB.Work )
   END_RUNG
   RUNG wire#powerrail
      I_Contact( #HMI.Selection[5] )
      R_Coil( #Fermi[5].DataIn.PB.Rest )
      R_Coil( #Fermi[5].DataIn.PB.Work )
   END_RUNG
   RUNG wire#powerrail
      I_Contact( #HMI.Selection[6] )
      R_Coil( #Fermi[6].DataIn.PB.Rest )
      R_Coil( #Fermi[6].DataIn.PB.Work )
   END_RUNG
   // the same network as SCL:
   IF NOT #HMI.Selection[1] THEN
       #Fermi[1].DataIn.PB.Rest := FALSE;
       #Fermi[1].DataIn.PB.Work := FALSE;
   END_IF;
   IF NOT #HMI.Selection[2] THEN
       #Fermi[2].DataIn.PB.Rest := FALSE;
       #Fermi[2].DataIn.PB.Work := FALSE;
   END_IF;
   IF NOT #HMI.Selection[3] THEN
       #Fermi[3].DataIn.PB.Rest := FALSE;
       #Fermi[3].DataIn.PB.Work := FALSE;
   END_IF;
   IF NOT #HMI.Selection[4] THEN
       #Fermi[4].DataIn.PB.Rest := FALSE;
       #Fermi[4].DataIn.PB.Work := FALSE;
   END_IF;
   IF NOT #HMI.Selection[5] THEN
       #Fermi[5].DataIn.PB.Rest := FALSE;
       #Fermi[5].DataIn.PB.Work := FALSE;
   END_IF;
   IF NOT #HMI.Selection[6] THEN
       #Fermi[6].DataIn.PB.Rest := FALSE;
       #Fermi[6].DataIn.PB.Work := FALSE;
   END_IF;
END_REGION

REGION Network 15: P[1...6] CIn External alarm
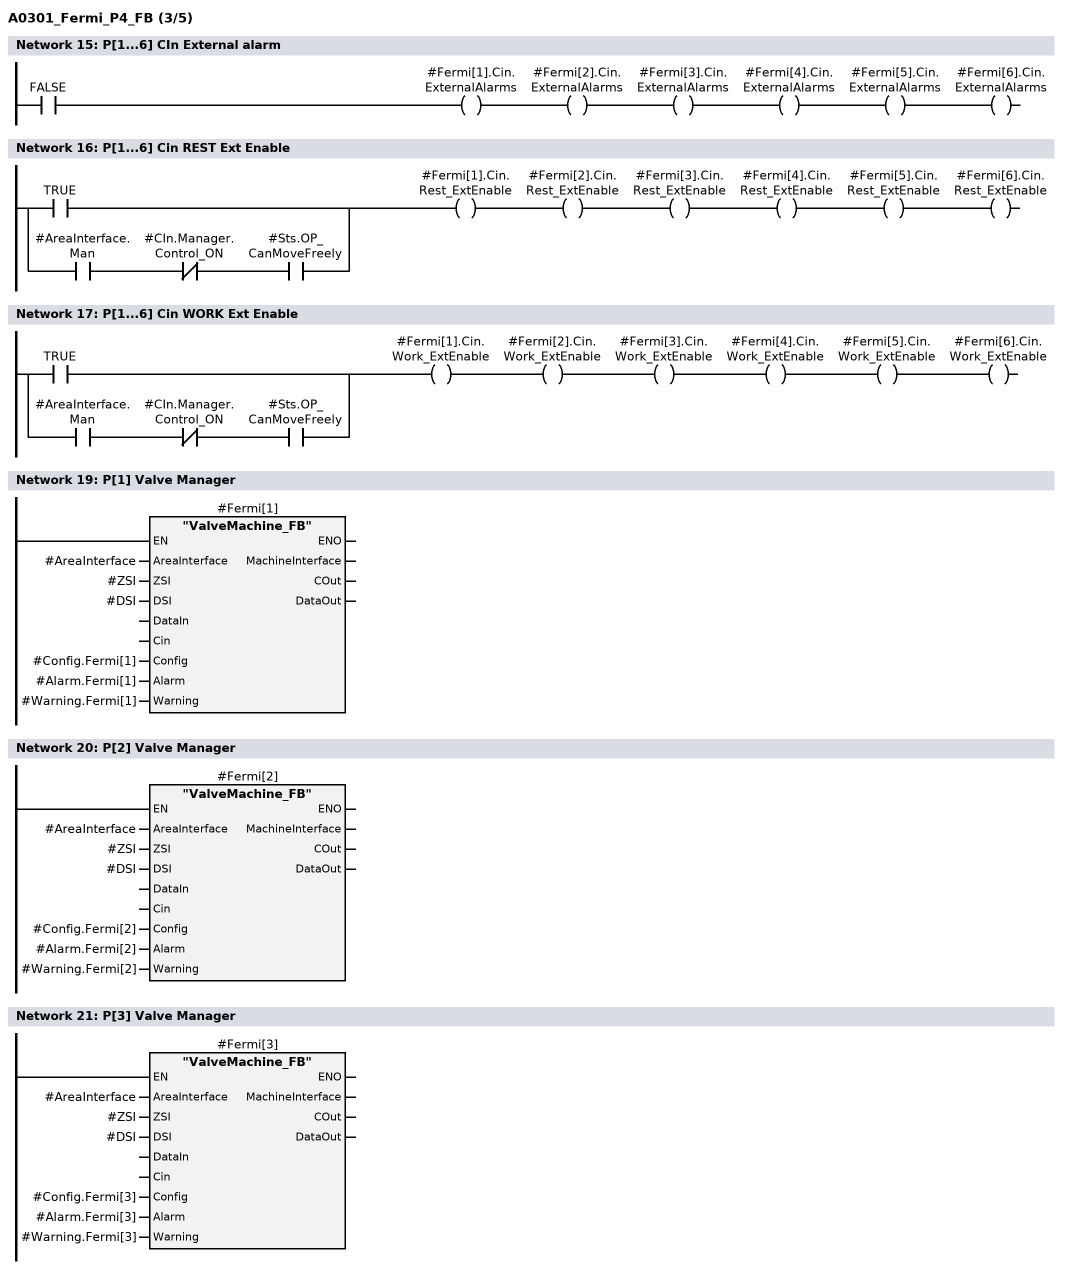
   RUNG wire#powerrail
      Contact( FALSE )
      Coil( #Fermi[1].Cin.ExternalAlarms )
      Coil( #Fermi[2].Cin.ExternalAlarms )
      Coil( #Fermi[3].Cin.ExternalAlarms )
      Coil( #Fermi[4].Cin.ExternalAlarms )
      Coil( #Fermi[5].Cin.ExternalAlarms )
      Coil( #Fermi[6].Cin.ExternalAlarms )
   END_RUNG
   // the same network as SCL:
   #Fermi[1].Cin.ExternalAlarms := FALSE;
   #Fermi[2].Cin.ExternalAlarms := FALSE;
   #Fermi[3].Cin.ExternalAlarms := FALSE;
   #Fermi[4].Cin.ExternalAlarms := FALSE;
   #Fermi[5].Cin.ExternalAlarms := FALSE;
   #Fermi[6].Cin.ExternalAlarms := FALSE;
END_REGION

REGION Network 16: P[1...6] Cin REST Ext Enable
   RUNG wire#powerrail
      Contact( TRUE )
      wire#w1
      Coil( #Fermi[1].Cin.Rest_ExtEnable )
      Coil( #Fermi[2].Cin.Rest_ExtEnable )
      Coil( #Fermi[3].Cin.Rest_ExtEnable )
      Coil( #Fermi[4].Cin.Rest_ExtEnable )
      Coil( #Fermi[5].Cin.Rest_ExtEnable )
      Coil( #Fermi[6].Cin.Rest_ExtEnable )
   END_RUNG
   RUNG wire#powerrail
      Contact( #AreaInterface.Man )
      I_Contact( #CIn.Manager.Control_ON )
      Contact( #Sts.OP_CanMoveFreely )
   END_RUNG wire#w1
   // the same network as SCL:
   #Fermi[1].Cin.Rest_ExtEnable := TRUE OR (#AreaInterface.Man AND NOT #CIn.Manager.Control_ON AND #Sts.OP_CanMoveFreely);
   #Fermi[2].Cin.Rest_ExtEnable := TRUE OR (#AreaInterface.Man AND NOT #CIn.Manager.Control_ON AND #Sts.OP_CanMoveFreely);
   #Fermi[3].Cin.Rest_ExtEnable := TRUE OR (#AreaInterface.Man AND NOT #CIn.Manager.Control_ON AND #Sts.OP_CanMoveFreely);
   #Fermi[4].Cin.Rest_ExtEnable := TRUE OR (#AreaInterface.Man AND NOT #CIn.Manager.Control_ON AND #Sts.OP_CanMoveFreely);
   #Fermi[5].Cin.Rest_ExtEnable := TRUE OR (#AreaInterface.Man AND NOT #CIn.Manager.Control_ON AND #Sts.OP_CanMoveFreely);
   #Fermi[6].Cin.Rest_ExtEnable := TRUE OR (#AreaInterface.Man AND NOT #CIn.Manager.Control_ON AND #Sts.OP_CanMoveFreely);
END_REGION

REGION Network 17: P[1...6] Cin WORK Ext Enable
   RUNG wire#powerrail
      Contact( TRUE )
      wire#w1
      Coil( #Fermi[1].Cin.Work_ExtEnable )
      Coil( #Fermi[2].Cin.Work_ExtEnable )
      Coil( #Fermi[3].Cin.Work_ExtEnable )
      Coil( #Fermi[4].Cin.Work_ExtEnable )
      Coil( #Fermi[5].Cin.Work_ExtEnable )
      Coil( #Fermi[6].Cin.Work_ExtEnable )
   END_RUNG
   RUNG wire#powerrail
      Contact( #AreaInterface.Man )
      I_Contact( #CIn.Manager.Control_ON )
      Contact( #Sts.OP_CanMoveFreely )
   END_RUNG wire#w1
   // the same network as SCL:
   #Fermi[1].Cin.Work_ExtEnable := TRUE OR (#AreaInterface.Man AND NOT #CIn.Manager.Control_ON AND #Sts.OP_CanMoveFreely);
   #Fermi[2].Cin.Work_ExtEnable := TRUE OR (#AreaInterface.Man AND NOT #CIn.Manager.Control_ON AND #Sts.OP_CanMoveFreely);
   #Fermi[3].Cin.Work_ExtEnable := TRUE OR (#AreaInterface.Man AND NOT #CIn.Manager.Control_ON AND #Sts.OP_CanMoveFreely);
   #Fermi[4].Cin.Work_ExtEnable := TRUE OR (#AreaInterface.Man AND NOT #CIn.Manager.Control_ON AND #Sts.OP_CanMoveFreely);
   #Fermi[5].Cin.Work_ExtEnable := TRUE OR (#AreaInterface.Man AND NOT #CIn.Manager.Control_ON AND #Sts.OP_CanMoveFreely);
   #Fermi[6].Cin.Work_ExtEnable := TRUE OR (#AreaInterface.Man AND NOT #CIn.Manager.Control_ON AND #Sts.OP_CanMoveFreely);
END_REGION

REGION Network 18: <+>
END_REGION

REGION Network 19: P[1] Valve Manager
   RUNG wire#powerrail
      #Fermi[1](AreaInterface := #AreaInterface, ZSI := #ZSI, DSI := #DSI, DataIn :=, Cin :=, Config := #Config.Fermi[1], Alarm := #Alarm.Fermi[1], Warning := #Warning.Fermi[1], MachineInterface =>, COut =>, DataOut =>)
   END_RUNG
   // the same network as SCL:
   #Fermi[1](AreaInterface := #AreaInterface,   // "ValveMachine_FB"
             ZSI := #ZSI,
             DSI := #DSI,
             Config := #Config.Fermi[1],
             Alarm := #Alarm.Fermi[1],
             Warning := #Warning.Fermi[1]);
END_REGION

REGION Network 20: P[2] Valve Manager
   RUNG wire#powerrail
      #Fermi[2](AreaInterface := #AreaInterface, ZSI := #ZSI, DSI := #DSI, DataIn :=, Cin :=, Config := #Config.Fermi[2], Alarm := #Alarm.Fermi[2], Warning := #Warning.Fermi[2], MachineInterface =>, COut =>, DataOut =>)
   END_RUNG
   // the same network as SCL:
   #Fermi[2](AreaInterface := #AreaInterface,   // "ValveMachine_FB"
             ZSI := #ZSI,
             DSI := #DSI,
             Config := #Config.Fermi[2],
             Alarm := #Alarm.Fermi[2],
             Warning := #Warning.Fermi[2]);
END_REGION

REGION Network 21: P[3] Valve Manager
   RUNG wire#powerrail
      #Fermi[3](AreaInterface := #AreaInterface, ZSI := #ZSI, DSI := #DSI, DataIn :=, Cin :=, Config := #Config.Fermi[3], Alarm := #Alarm.Fermi[3], Warning := #Warning.Fermi[3], MachineInterface =>, COut =>, DataOut =>)
   END_RUNG
   // the same network as SCL:
   #Fermi[3](AreaInterface := #AreaInterface,   // "ValveMachine_FB"
             ZSI := #ZSI,
             DSI := #DSI,
             Config := #Config.Fermi[3],
             Alarm := #Alarm.Fermi[3],
             Warning := #Warning.Fermi[3]);
END_REGION

REGION Network 22: P[4] Valve Manager
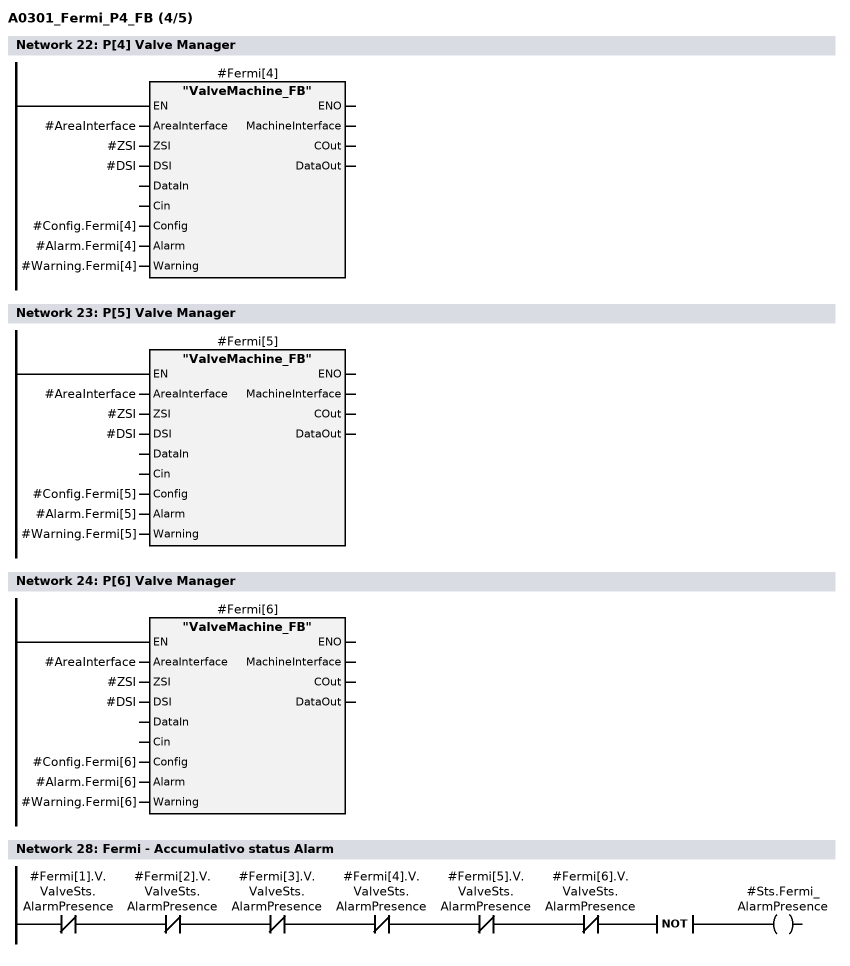
   RUNG wire#powerrail
      #Fermi[4](AreaInterface := #AreaInterface, ZSI := #ZSI, DSI := #DSI, DataIn :=, Cin :=, Config := #Config.Fermi[4], Alarm := #Alarm.Fermi[4], Warning := #Warning.Fermi[4], MachineInterface =>, COut =>, DataOut =>)
   END_RUNG
   // the same network as SCL:
   #Fermi[4](AreaInterface := #AreaInterface,   // "ValveMachine_FB"
             ZSI := #ZSI,
             DSI := #DSI,
             Config := #Config.Fermi[4],
             Alarm := #Alarm.Fermi[4],
             Warning := #Warning.Fermi[4]);
END_REGION

REGION Network 23: P[5] Valve Manager
   RUNG wire#powerrail
      #Fermi[5](AreaInterface := #AreaInterface, ZSI := #ZSI, DSI := #DSI, DataIn :=, Cin :=, Config := #Config.Fermi[5], Alarm := #Alarm.Fermi[5], Warning := #Warning.Fermi[5], MachineInterface =>, COut =>, DataOut =>)
   END_RUNG
   // the same network as SCL:
   #Fermi[5](AreaInterface := #AreaInterface,   // "ValveMachine_FB"
             ZSI := #ZSI,
             DSI := #DSI,
             Config := #Config.Fermi[5],
             Alarm := #Alarm.Fermi[5],
             Warning := #Warning.Fermi[5]);
END_REGION

REGION Network 24: P[6] Valve Manager
   RUNG wire#powerrail
      #Fermi[6](AreaInterface := #AreaInterface, ZSI := #ZSI, DSI := #DSI, DataIn :=, Cin :=, Config := #Config.Fermi[6], Alarm := #Alarm.Fermi[6], Warning := #Warning.Fermi[6], MachineInterface =>, COut =>, DataOut =>)
   END_RUNG
   // the same network as SCL:
   #Fermi[6](AreaInterface := #AreaInterface,   // "ValveMachine_FB"
             ZSI := #ZSI,
             DSI := #DSI,
             Config := #Config.Fermi[6],
             Alarm := #Alarm.Fermi[6],
             Warning := #Warning.Fermi[6]);
END_REGION

REGION Network 25: <+>
END_REGION

REGION Network 26 (SCL): P[1...6] COut Fermi
   REGION COut STANDSTILL Fermi
       // Controllo uscita COut STANDSTILL in base allo stato di tutti i Pin
       IF  #Fermi[1].Sts.Standstill AND
           #Fermi[2].Sts.Standstill AND
           #Fermi[3].Sts.Standstill AND
           #Fermi[4].Sts.Standstill AND
           #Fermi[5].Sts.Standstill AND
           #Fermi[6].Sts.Standstill THEN
           #COut.Fermi.Standstill := TRUE;
       ELSE
           #COut.Fermi.Standstill := FALSE;
       END_IF;
   END_REGION ;

   REGION COut AT REST #Fermi
       // Controllo uscita COut AT_REST in base allo stato di tutti i Pin
       IF  #Fermi[1].COut.Rest OR #Fermi[1].DataIn.Rest_Ls[1] AND
           #Fermi[2].COut.Rest OR #Fermi[2].DataIn.Rest_Ls[1] AND
           #Fermi[3].COut.Rest OR #Fermi[3].DataIn.Rest_Ls[1] AND
           #Fermi[4].COut.Rest OR #Fermi[4].DataIn.Rest_Ls[1] AND
           #Fermi[5].COut.Rest OR #Fermi[5].DataIn.Rest_Ls[1] AND
           #Fermi[6].COut.Rest OR #Fermi[6].DataIn.Rest_Ls[1] THEN
           #COut.Fermi.Rest := 1;
       ELSE
           #COut.Fermi.Rest := 0;
       END_IF;
   END_REGION ;

   REGION COut AT WORK Fermi
       // Controllo uscita COut AT_WORK in base allo stato di tutti i Pin
       IF #Fermi[1].COut.Work AND
           #Fermi[2].COut.Work AND
           #Fermi[3].COut.Work AND
           #Fermi[4].COut.Work AND
           #Fermi[5].COut.Work AND
           #Fermi[6].COut.Work THEN
           #COut.Fermi.Work := 1;
       ELSE
           #COut.Fermi.Work := 0;
       END_IF;
   END_REGION ;
END_REGION

REGION Network 28: Fermi - Accumulativo status Alarm
   RUNG wire#powerrail
      I_Contact( #Fermi[1].V.ValveSts.AlarmPresence )
      I_Contact( #Fermi[2].V.ValveSts.AlarmPresence )
      I_Contact( #Fermi[3].V.ValveSts.AlarmPresence )
      I_Contact( #Fermi[4].V.ValveSts.AlarmPresence )
      I_Contact( #Fermi[5].V.ValveSts.AlarmPresence )
      I_Contact( #Fermi[6].V.ValveSts.AlarmPresence )
      Not()
      Coil( #Sts.Fermi_AlarmPresence )
   END_RUNG
   // the same network as SCL:
   #Sts.Fermi_AlarmPresence := NOT (NOT #Fermi[1].V.ValveSts.AlarmPresence AND NOT #Fermi[2].V.ValveSts.AlarmPresence AND NOT #Fermi[3].V.ValveSts.AlarmPresence AND NOT #Fermi[4].V.ValveSts.AlarmPresence AND NOT #Fermi[5].V.ValveSts.AlarmPresence AND NOT #Fermi[6].V.ValveSts.AlarmPresence);
END_REGION

REGION Network 29 (SCL): HMI STATUS - Postazione
   // Area dati appoggio per HMI
   // FERMI POS.3
   #HMI.FermiSts.Standstill := #COut.Fermi.Standstill;
   #HMI.FermiSts.Rest := #COut.Fermi.Rest;
   #HMI.FermiSts.Work := #COut.Fermi.Work;
   #HMI.FermiSts.AlarmPresence := #Sts.Fermi_AlarmPresence;
END_REGION

REGION Network 31: << MAIN MACHINE STATUS >>
END_REGION

REGION Network 32: Machine interface
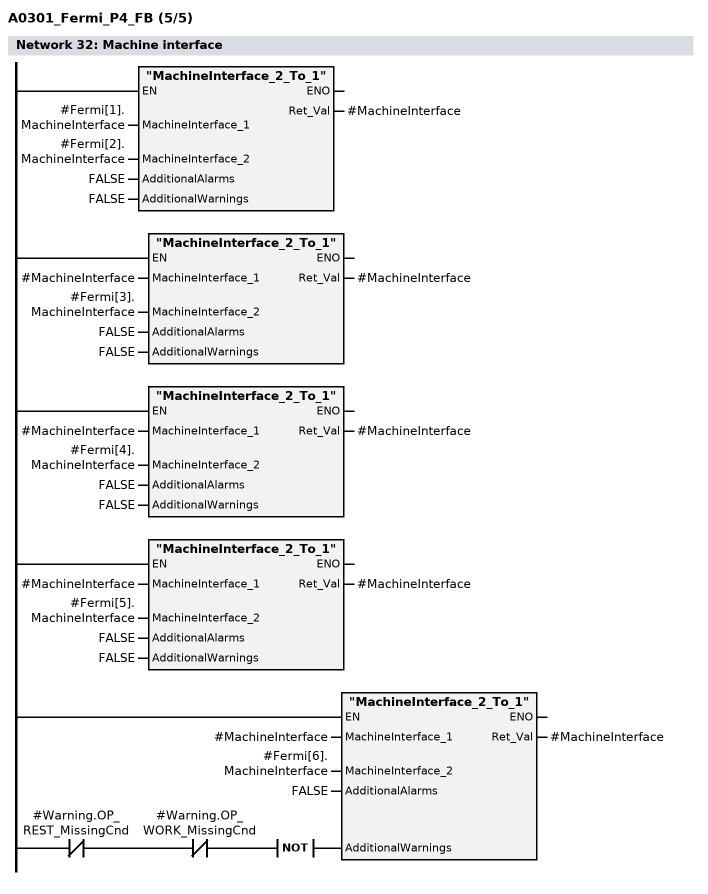
   RUNG wire#powerrail
      "MachineInterface_2_To_1"(MachineInterface_1 := #Fermi[1].MachineInterface, MachineInterface_2 := #Fermi[2].MachineInterface, AdditionalAlarms := FALSE, AdditionalWarnings := FALSE, Ret_Val => #MachineInterface)
   END_RUNG
   RUNG wire#powerrail
      "MachineInterface_2_To_1"(MachineInterface_1 := #MachineInterface, MachineInterface_2 := #Fermi[3].MachineInterface, AdditionalAlarms := FALSE, AdditionalWarnings := FALSE, Ret_Val => #MachineInterface)
   END_RUNG
   RUNG wire#powerrail
      "MachineInterface_2_To_1"(MachineInterface_1 := #MachineInterface, MachineInterface_2 := #Fermi[4].MachineInterface, AdditionalAlarms := FALSE, AdditionalWarnings := FALSE, Ret_Val => #MachineInterface)
   END_RUNG
   RUNG wire#powerrail
      "MachineInterface_2_To_1"(MachineInterface_1 := #MachineInterface, MachineInterface_2 := #Fermi[5].MachineInterface, AdditionalAlarms := FALSE, AdditionalWarnings := FALSE, Ret_Val => #MachineInterface)
   END_RUNG
   RUNG wire#powerrail
      "MachineInterface_2_To_1"(AdditionalWarnings := wire#w1, MachineInterface_1 := #MachineInterface, MachineInterface_2 := #Fermi[6].MachineInterface, AdditionalAlarms := FALSE, Ret_Val => #MachineInterface)
   END_RUNG
   RUNG wire#powerrail
      I_Contact( #Warning.OP_REST_MissingCnd )
      I_Contact( #Warning.OP_WORK_MissingCnd )
      Not()
   END_RUNG wire#w1
   // the same network as SCL:
   #MachineInterface := "MachineInterface_2_To_1"(MachineInterface_1 := #Fermi[1].MachineInterface,
                           MachineInterface_2 := #Fermi[2].MachineInterface,
                           AdditionalAlarms := FALSE,
                           AdditionalWarnings := FALSE);
   #MachineInterface := "MachineInterface_2_To_1"(MachineInterface_1 := #MachineInterface,
                           MachineInterface_2 := #Fermi[3].MachineInterface,
                           AdditionalAlarms := FALSE,
                           AdditionalWarnings := FALSE);
   #MachineInterface := "MachineInterface_2_To_1"(MachineInterface_1 := #MachineInterface,
                           MachineInterface_2 := #Fermi[4].MachineInterface,
                           AdditionalAlarms := FALSE,
                           AdditionalWarnings := FALSE);
   #MachineInterface := "MachineInterface_2_To_1"(MachineInterface_1 := #MachineInterface,
                           MachineInterface_2 := #Fermi[5].MachineInterface,
                           AdditionalAlarms := FALSE,
                           AdditionalWarnings := FALSE);
   #MachineInterface := "MachineInterface_2_To_1"(MachineInterface_1 := #MachineInterface,
                           MachineInterface_2 := #Fermi[6].MachineInterface,
                           AdditionalAlarms := FALSE,
                           AdditionalWarnings := NOT (NOT #Warning.OP_REST_MissingCnd AND NOT #Warning.OP_WORK_MissingCnd));
END_REGION
END_FUNCTION_BLOCK

FUNCTION "A0301_Spintore_Lat_CALL" : Void   // FC3, LAD
TITLE = <<< SPINTORE LATERALE 1 >>>
// stored: SetENOAutomatically false
BEGIN

REGION Network 1 (SCL): << TRASFERIMENTO stati CIn del blocco >>
   REGION TRASFERIMENTO CIn MANAGER
       "A0301_Spintore_Lat".CIn.Manager_SpinLat_1 := "A0301_Manager".COut.P5.Spintore_Lat_1;
       "A0301_Spintore_Lat".CIn.Manager_SpinLat_2 := "A0301_Manager".COut.P5.Spintore_Lat_2;
       "A0301_Spintore_Lat".CIn.Manager_Sollevatori := "A0301_Manager".COut.P5.Sollevatori;
       //
       "A0301_Spintore_Lat".CIn.SemiAut_Pb := "A0301_Manager".DataIn.SemiAut_Pb;
   END_REGION ;

   REGION TRASFERIMENTO CIn FERMI POSTAZIONI P4/P5, DEI FERMI SU P4 E DEI SOLLEVATORI SU P5 
       // Trasferimento status alla Stazione Spintore Laterale 1 da COut a Cin della P4
       "A0301_Spintore_Lat".CIn.P4.Fermi := "A0301_Fermi_P4".COut.Fermi;
   END_REGION ;

   REGION TRASFERIMENTO CIn POSTAZIONI P5
       // Trasferimento status alla Stazione Spintore Laterale 1 da COut a Cin della P4
       "A0301_Spintore_Lat".CIn.P5.SpintoreLong.Ax := "A0302_Spintore".COut.Ax;
       "A0301_Spintore_Lat".CIn.P5.SpintoreLong.Ax_Sts:= "A0302_Spintore".COut.Ax_Sts;
       "A0301_Spintore_Lat".CIn.P5.SpintoreLong.Spintore:= "A0302_Spintore".COut.Spintore;
       "A0301_Spintore_Lat".CIn.P5.SpintoreLong.Vrt:= "A0302_Spintore".COut.Vrt;
       "A0301_Spintore_Lat".CIn.P5.SpintoreLong.Orz:= "A0302_Spintore".COut.Orz;

   END_REGION ;

   REGION TRASFERIMENTO CIn TRASPORTO 
       // Trasferimenti status lettura posizioni Trasporto al Cin delle stazioni
       "A0301_Spintore_Lat".CIn.Trasporto := "A0301_Trasporto".COut.Ax;
   END_REGION ;

   // Trasferimento BTrk della larghezza dei Beams
   "A0301_Spintore_Lat".Sts.Beam.H_B := "BTrk".A0301.Beam_H_B;
   "A0301_Spintore_Lat".Sts.Beam.Len_Meas := "A0302_Spintore".Sts.A0302_Beam_BLean;
END_REGION

REGION Network 2 (SCL): << TRASFERIMENTO stati DataIn >>
   REGION TRASFERIMENTO #DataIn STATI OPERATION BUTTON STAZIONE SPINTORE LATERALE 
       // PB FERMI VERTICALI
       "A0301_Spintore_Lat".DataIn.OP_Rest_PB := "A03_HMI".MB3.Button.A0301.SpintoreLat.OP.Rest;
       "A0301_Spintore_Lat".DataIn.OP_Work_PB := "A03_HMI".MB3.Button.A0301.SpintoreLat.OP.Work;
   END_REGION ;

   REGION TRASFERIMENTO STATO LETTURA SENSORI DELLA STAZIONE SPINTORE LATERALE
       // Ingresso analogico di controllo Work Pos. Spintore Orizzontale
       "A0301_Spintore_Lat".DataIn.Orz_1_AnalSens:= "A0302_AI_SpintoreLaterale_1_Posizionamento";
       "A0301_Spintore_Lat".DataIn.Orz_2_AnalSens := "A0302_AI_SpintoreLaterale_2_Posizionamento";

   END_REGION ;
END_REGION

REGION Network 3: << Data In PB - Spintori Vertivale >>
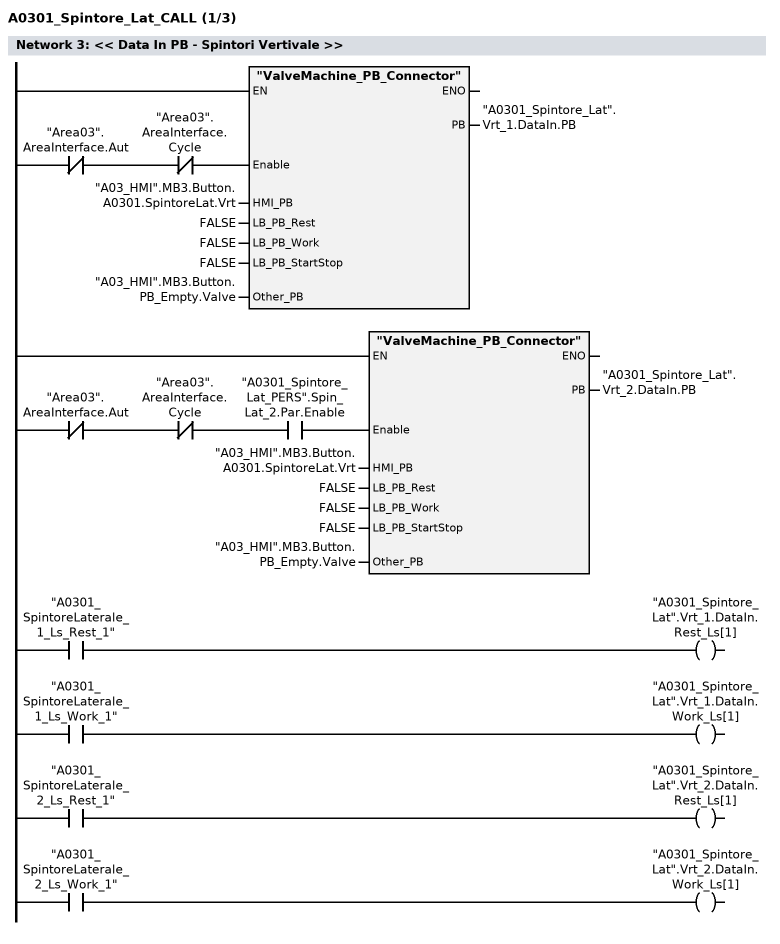
   RUNG wire#powerrail
      "ValveMachine_PB_Connector"(Enable := wire#w1, HMI_PB := "A03_HMI".MB3.Button.A0301.SpintoreLat.Vrt, LB_PB_Rest := FALSE, LB_PB_Work := FALSE, LB_PB_StartStop := FALSE, Other_PB := "A03_HMI".MB3.Button.PB_Empty.Valve, PB => "A0301_Spintore_Lat".Vrt_1.DataIn.PB)
   END_RUNG
   RUNG wire#powerrail
      I_Contact( "Area03".AreaInterface.Aut )
      I_Contact( "Area03".AreaInterface.Cycle )
   END_RUNG wire#w1
   RUNG wire#powerrail
      "ValveMachine_PB_Connector"(Enable := wire#w2, HMI_PB := "A03_HMI".MB3.Button.A0301.SpintoreLat.Vrt, LB_PB_Rest := FALSE, LB_PB_Work := FALSE, LB_PB_StartStop := FALSE, Other_PB := "A03_HMI".MB3.Button.PB_Empty.Valve, PB => "A0301_Spintore_Lat".Vrt_2.DataIn.PB)
   END_RUNG
   RUNG wire#powerrail
      I_Contact( "Area03".AreaInterface.Aut )
      I_Contact( "Area03".AreaInterface.Cycle )
      Contact( "A0301_Spintore_Lat_PERS".Spin_Lat_2.Par.Enable )
   END_RUNG wire#w2
   RUNG wire#powerrail
      Contact( "A0301_SpintoreLaterale_1_Ls_Rest_1" )
      Coil( "A0301_Spintore_Lat".Vrt_1.DataIn.Rest_Ls[1] )
   END_RUNG
   RUNG wire#powerrail
      Contact( "A0301_SpintoreLaterale_1_Ls_Work_1" )
      Coil( "A0301_Spintore_Lat".Vrt_1.DataIn.Work_Ls[1] )
   END_RUNG
   RUNG wire#powerrail
      Contact( "A0301_SpintoreLaterale_2_Ls_Rest_1" )
      Coil( "A0301_Spintore_Lat".Vrt_2.DataIn.Rest_Ls[1] )
   END_RUNG
   RUNG wire#powerrail
      Contact( "A0301_SpintoreLaterale_2_Ls_Work_1" )
      Coil( "A0301_Spintore_Lat".Vrt_2.DataIn.Work_Ls[1] )
   END_RUNG
   // the same network as SCL:
   "ValveMachine_PB_Connector"(Enable := NOT "Area03".AreaInterface.Aut AND NOT "Area03".AreaInterface.Cycle,
                           HMI_PB := "A03_HMI".MB3.Button.A0301.SpintoreLat.Vrt,
                           LB_PB_Rest := FALSE,
                           LB_PB_Work := FALSE,
                           LB_PB_StartStop := FALSE,
                           Other_PB := "A03_HMI".MB3.Button.PB_Empty.Valve,
                           PB => "A0301_Spintore_Lat".Vrt_1.DataIn.PB);
   "ValveMachine_PB_Connector"(Enable := NOT "Area03".AreaInterface.Aut AND NOT "Area03".AreaInterface.Cycle AND "A0301_Spintore_Lat_PERS".Spin_Lat_2.Par.Enable,
                           HMI_PB := "A03_HMI".MB3.Button.A0301.SpintoreLat.Vrt,
                           LB_PB_Rest := FALSE,
                           LB_PB_Work := FALSE,
                           LB_PB_StartStop := FALSE,
                           Other_PB := "A03_HMI".MB3.Button.PB_Empty.Valve,
                           PB => "A0301_Spintore_Lat".Vrt_2.DataIn.PB);
   "A0301_Spintore_Lat".Vrt_1.DataIn.Rest_Ls[1] := "A0301_SpintoreLaterale_1_Ls_Rest_1";
   "A0301_Spintore_Lat".Vrt_1.DataIn.Work_Ls[1] := "A0301_SpintoreLaterale_1_Ls_Work_1";
   "A0301_Spintore_Lat".Vrt_2.DataIn.Rest_Ls[1] := "A0301_SpintoreLaterale_2_Ls_Rest_1";
   "A0301_Spintore_Lat".Vrt_2.DataIn.Work_Ls[1] := "A0301_SpintoreLaterale_2_Ls_Work_1";
END_REGION

REGION Network 4: << Data In PB - Spintore Orizzontale >>
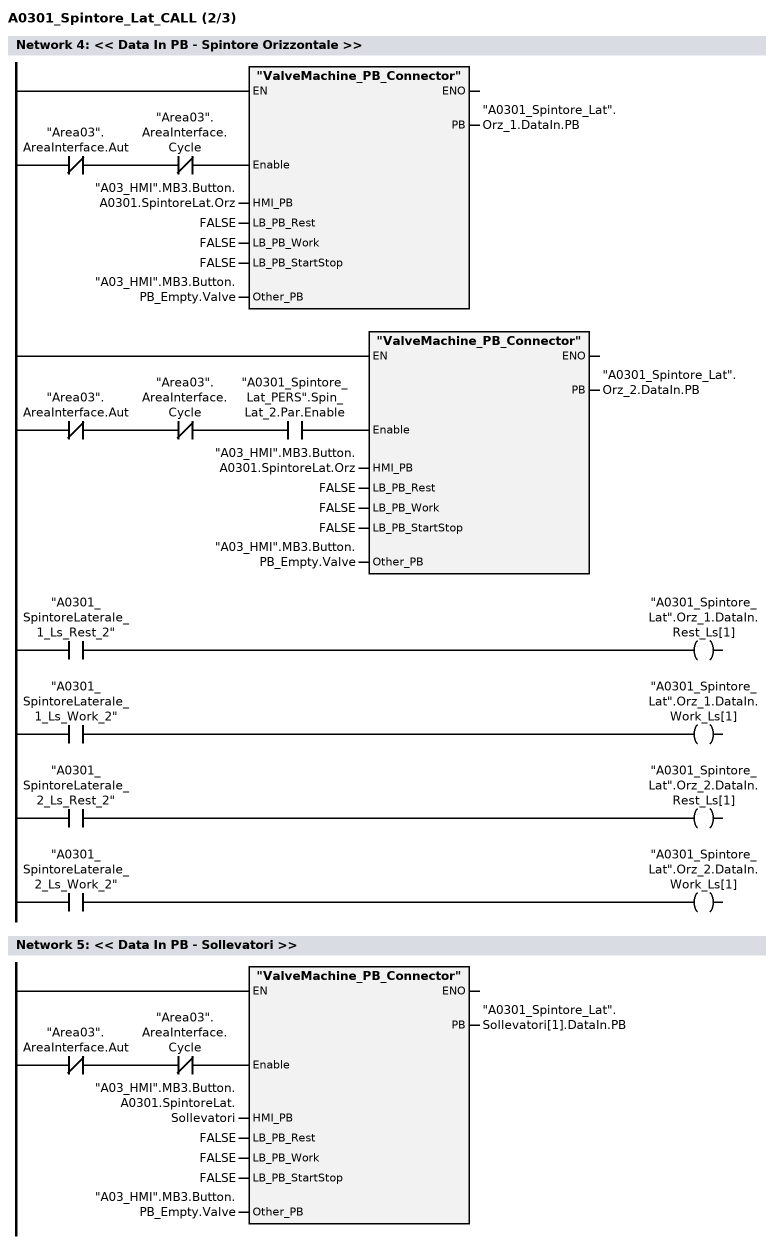
   RUNG wire#powerrail
      "ValveMachine_PB_Connector"(Enable := wire#w1, HMI_PB := "A03_HMI".MB3.Button.A0301.SpintoreLat.Orz, LB_PB_Rest := FALSE, LB_PB_Work := FALSE, LB_PB_StartStop := FALSE, Other_PB := "A03_HMI".MB3.Button.PB_Empty.Valve, PB => "A0301_Spintore_Lat".Orz_1.DataIn.PB)
   END_RUNG
   RUNG wire#powerrail
      I_Contact( "Area03".AreaInterface.Aut )
      I_Contact( "Area03".AreaInterface.Cycle )
   END_RUNG wire#w1
   RUNG wire#powerrail
      "ValveMachine_PB_Connector"(Enable := wire#w2, HMI_PB := "A03_HMI".MB3.Button.A0301.SpintoreLat.Orz, LB_PB_Rest := FALSE, LB_PB_Work := FALSE, LB_PB_StartStop := FALSE, Other_PB := "A03_HMI".MB3.Button.PB_Empty.Valve, PB => "A0301_Spintore_Lat".Orz_2.DataIn.PB)
   END_RUNG
   RUNG wire#powerrail
      I_Contact( "Area03".AreaInterface.Aut )
      I_Contact( "Area03".AreaInterface.Cycle )
      Contact( "A0301_Spintore_Lat_PERS".Spin_Lat_2.Par.Enable )
   END_RUNG wire#w2
   RUNG wire#powerrail
      Contact( "A0301_SpintoreLaterale_1_Ls_Rest_2" )
      Coil( "A0301_Spintore_Lat".Orz_1.DataIn.Rest_Ls[1] )
   END_RUNG
   RUNG wire#powerrail
      Contact( "A0301_SpintoreLaterale_1_Ls_Work_2" )
      Coil( "A0301_Spintore_Lat".Orz_1.DataIn.Work_Ls[1] )
   END_RUNG
   RUNG wire#powerrail
      Contact( "A0301_SpintoreLaterale_2_Ls_Rest_2" )
      Coil( "A0301_Spintore_Lat".Orz_2.DataIn.Rest_Ls[1] )
   END_RUNG
   RUNG wire#powerrail
      Contact( "A0301_SpintoreLaterale_2_Ls_Work_2" )
      Coil( "A0301_Spintore_Lat".Orz_2.DataIn.Work_Ls[1] )
   END_RUNG
   // the same network as SCL:
   "ValveMachine_PB_Connector"(Enable := NOT "Area03".AreaInterface.Aut AND NOT "Area03".AreaInterface.Cycle,
                           HMI_PB := "A03_HMI".MB3.Button.A0301.SpintoreLat.Orz,
                           LB_PB_Rest := FALSE,
                           LB_PB_Work := FALSE,
                           LB_PB_StartStop := FALSE,
                           Other_PB := "A03_HMI".MB3.Button.PB_Empty.Valve,
                           PB => "A0301_Spintore_Lat".Orz_1.DataIn.PB);
   "ValveMachine_PB_Connector"(Enable := NOT "Area03".AreaInterface.Aut AND NOT "Area03".AreaInterface.Cycle AND "A0301_Spintore_Lat_PERS".Spin_Lat_2.Par.Enable,
                           HMI_PB := "A03_HMI".MB3.Button.A0301.SpintoreLat.Orz,
                           LB_PB_Rest := FALSE,
                           LB_PB_Work := FALSE,
                           LB_PB_StartStop := FALSE,
                           Other_PB := "A03_HMI".MB3.Button.PB_Empty.Valve,
                           PB => "A0301_Spintore_Lat".Orz_2.DataIn.PB);
   "A0301_Spintore_Lat".Orz_1.DataIn.Rest_Ls[1] := "A0301_SpintoreLaterale_1_Ls_Rest_2";
   "A0301_Spintore_Lat".Orz_1.DataIn.Work_Ls[1] := "A0301_SpintoreLaterale_1_Ls_Work_2";
   "A0301_Spintore_Lat".Orz_2.DataIn.Rest_Ls[1] := "A0301_SpintoreLaterale_2_Ls_Rest_2";
   "A0301_Spintore_Lat".Orz_2.DataIn.Work_Ls[1] := "A0301_SpintoreLaterale_2_Ls_Work_2";
END_REGION

REGION Network 5: << Data In PB - Sollevatori >>
   RUNG wire#powerrail
      "ValveMachine_PB_Connector"(Enable := wire#w1, HMI_PB := "A03_HMI".MB3.Button.A0301.SpintoreLat.Sollevatori, LB_PB_Rest := FALSE, LB_PB_Work := FALSE, LB_PB_StartStop := FALSE, Other_PB := "A03_HMI".MB3.Button.PB_Empty.Valve, PB => "A0301_Spintore_Lat".Sollevatori[1].DataIn.PB)
   END_RUNG
   RUNG wire#powerrail
      I_Contact( "Area03".AreaInterface.Aut )
      I_Contact( "Area03".AreaInterface.Cycle )
   END_RUNG wire#w1
   // the same network as SCL:
   "ValveMachine_PB_Connector"(Enable := NOT "Area03".AreaInterface.Aut AND NOT "Area03".AreaInterface.Cycle,
                           HMI_PB := "A03_HMI".MB3.Button.A0301.SpintoreLat.Sollevatori,
                           LB_PB_Rest := FALSE,
                           LB_PB_Work := FALSE,
                           LB_PB_StartStop := FALSE,
                           Other_PB := "A03_HMI".MB3.Button.PB_Empty.Valve,
                           PB => "A0301_Spintore_Lat".Sollevatori[1].DataIn.PB);
END_REGION

REGION Network 6 (SCL): DataIn - Ls Sollevatori [1..6]
   // Ls Riposo
   "A0301_Spintore_Lat".Sollevatori[1].DataIn.Rest_Ls[1] := "A0301_CinghiaTrasporto_1.2_Ls_Rest_5";
   "A0301_Spintore_Lat".Sollevatori[2].DataIn.Rest_Ls[1] := "A0301_CinghiaTrasporto_2.2_Ls_Rest_5";
   "A0301_Spintore_Lat".Sollevatori[3].DataIn.Rest_Ls[1] := "A0301_CinghiaTrasporto_3.2_Ls_Rest_5";
   "A0301_Spintore_Lat".Sollevatori[4].DataIn.Rest_Ls[1] := "A0301_CinghiaTrasporto_4.2_Ls_Rest_5";
   "A0301_Spintore_Lat".Sollevatori[5].DataIn.Rest_Ls[1] := "A0301_CinghiaTrasporto_5.2_Ls_Rest_5";
   "A0301_Spintore_Lat".Sollevatori[6].DataIn.Rest_Ls[1] := "A0301_CinghiaTrasporto_6.2_Ls_Rest_5";
END_REGION

REGION Network 7 (SCL): DataIn - PB Sollevatori [1..6]
   // TRASFERIMENTO STATO PULSANTI - Comando manuale diretto
   "A0301_Spintore_Lat".Sollevatori[6].DataIn.PB:="A0301_Spintore_Lat".Sollevatori[5].DataIn.PB:=
   "A0301_Spintore_Lat".Sollevatori[4].DataIn.PB := "A0301_Spintore_Lat".Sollevatori[3].DataIn.PB :=
   "A0301_Spintore_Lat".Sollevatori[2].DataIn.PB:= "A0301_Spintore_Lat".Sollevatori[1].DataIn.PB;
END_REGION

REGION Network 8: <+>
END_REGION

REGION Network 9: [Spintore Laterale] - Machine Call
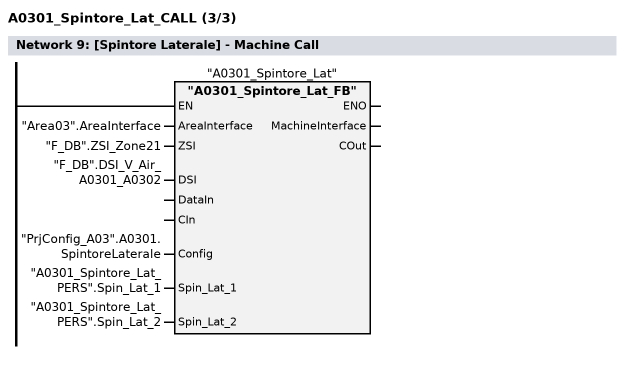
   RUNG wire#powerrail
      "A0301_Spintore_Lat"(AreaInterface := "Area03".AreaInterface, ZSI := "F_DB".ZSI_Zone21, DSI := "F_DB".DSI_V_Air_A0301_A0302, DataIn :=, CIn :=, Config := "PrjConfig_A03".A0301.SpintoreLaterale, Spin_Lat_1 := "A0301_Spintore_Lat_PERS".Spin_Lat_1, Spin_Lat_2 := "A0301_Spintore_Lat_PERS".Spin_Lat_2, MachineInterface =>, COut =>)
   END_RUNG
   // the same network as SCL:
   "A0301_Spintore_Lat"(AreaInterface := "Area03".AreaInterface,   // "A0301_Spintore_Lat_FB"
                        ZSI := "F_DB".ZSI_Zone21,
                        DSI := "F_DB".DSI_V_Air_A0301_A0302,
                        Config := "PrjConfig_A03".A0301.SpintoreLaterale,
                        Spin_Lat_1 := "A0301_Spintore_Lat_PERS".Spin_Lat_1,
                        Spin_Lat_2 := "A0301_Spintore_Lat_PERS".Spin_Lat_2);
END_REGION

REGION Network 10 (SCL): << TRASFERIMENTO stati DataOut >>
   REGION COMANDO DELLE USCITE SPINTORE LATERALE 1 & 2

       // Fermi Verticali blocco prodotto SPINTORE LATERALE 1 - RIPOSO
       "A0301_SpintoreLaterale_1_V_Rest_1" := "A0301_Spintore_Lat".Vrt_1.DataOut.RestSolenoid;

       // Fermi Verticali blocco prodotto Stazione SPINTORE LATERALE 1 - LAVORO
       "A0301_SpintoreLaterale_1_V_Work_1" := "A0301_Spintore_Lat".Vrt_1.DataOut.WorkSolenoid;

       // Spintore Orizzontale trasla prodotto SPINTORE LATERALE 1 - RIPOSO
       "A0301_SpintoreLaterale_1_V_Rest_2" := "A0301_Spintore_Lat".Orz_1.DataOut.RestSolenoid;

       // Spintore Orizzontale trasla prodotto SPINTORE LATERALE 1 - LAVORO
       "A0301_SpintoreLaterale_1_V_Work_2" := "A0301_Spintore_Lat".Orz_1.DataOut.WorkSolenoid;

       // ***************************************************************************************    
       // Fermi Verticali blocco prodotto SPINTORE LATERALE 2 - RIPOSO

       "A0301_SpintoreLaterale_2_V_Rest_1" := "A0301_Spintore_Lat".Vrt_2.DataOut.RestSolenoid;

       // Fermi Verticali blocco prodotto Stazione SPINTORE LATERALE 2 - LAVORO

       "A0301_SpintoreLaterale_2_V_Work_1" := "A0301_Spintore_Lat".Vrt_2.DataOut.WorkSolenoid;

       // Spintore Orizzontale trasla prodotto SPINTORE LATERALE 2 - RIPOSO

       "A0301_SpintoreLaterale_2_V_Rest_2" := "A0301_Spintore_Lat".Orz_2.DataOut.RestSolenoid;

       // Spintore Orizzontale trasla prodotto SPINTORE LATERALE 2 - LAVORO

       "A0301_SpintoreLaterale_2_V_Work_2" := "A0301_Spintore_Lat".Orz_2.DataOut.WorkSolenoid;


   END_REGION ;

   REGION COMANDO USCITE SOLLEVATORI P5
       "A0301_CinghiaTrasporto_1.2_V_Rest_5" := "A0301_Spintore_Lat".Sollevatori[1].DataOut.RestSolenoid;
       "A0301_CinghiaTrasporto_2.2_V_Rest_5" := "A0301_Spintore_Lat".Sollevatori[2].DataOut.RestSolenoid;
       "A0301_CinghiaTrasporto_3.2_V_Rest_5" := "A0301_Spintore_Lat".Sollevatori[3].DataOut.RestSolenoid;
       "A0301_CinghiaTrasporto_4.2_V_Rest_5" := "A0301_Spintore_Lat".Sollevatori[4].DataOut.RestSolenoid;
       "A0301_CinghiaTrasporto_5.2_V_Rest_5" := "A0301_Spintore_Lat".Sollevatori[5].DataOut.RestSolenoid;
       "A0301_CinghiaTrasporto_6.2_V_Rest_5" := "A0301_Spintore_Lat".Sollevatori[6].DataOut.RestSolenoid;


       "A0301_CinghiaTrasporto_1.2_V_Work_6" := "A0301_Spintore_Lat".Sollevatori[1].DataOut.WorkSolenoid;
       "A0301_CinghiaTrasporto_2.2_V_Work_6" := "A0301_Spintore_Lat".Sollevatori[2].DataOut.WorkSolenoid;
       "A0301_CinghiaTrasporto_3.2_V_Work_6" := "A0301_Spintore_Lat".Sollevatori[3].DataOut.WorkSolenoid;
       "A0301_CinghiaTrasporto_4.2_V_Work_6" := "A0301_Spintore_Lat".Sollevatori[4].DataOut.WorkSolenoid;
       "A0301_CinghiaTrasporto_5.2_V_Work_6" := "A0301_Spintore_Lat".Sollevatori[5].DataOut.WorkSolenoid;
       "A0301_CinghiaTrasporto_6.2_V_Work_6" := "A0301_Spintore_Lat".Sollevatori[6].DataOut.WorkSolenoid;


   END_REGION
END_REGION
END_FUNCTION

